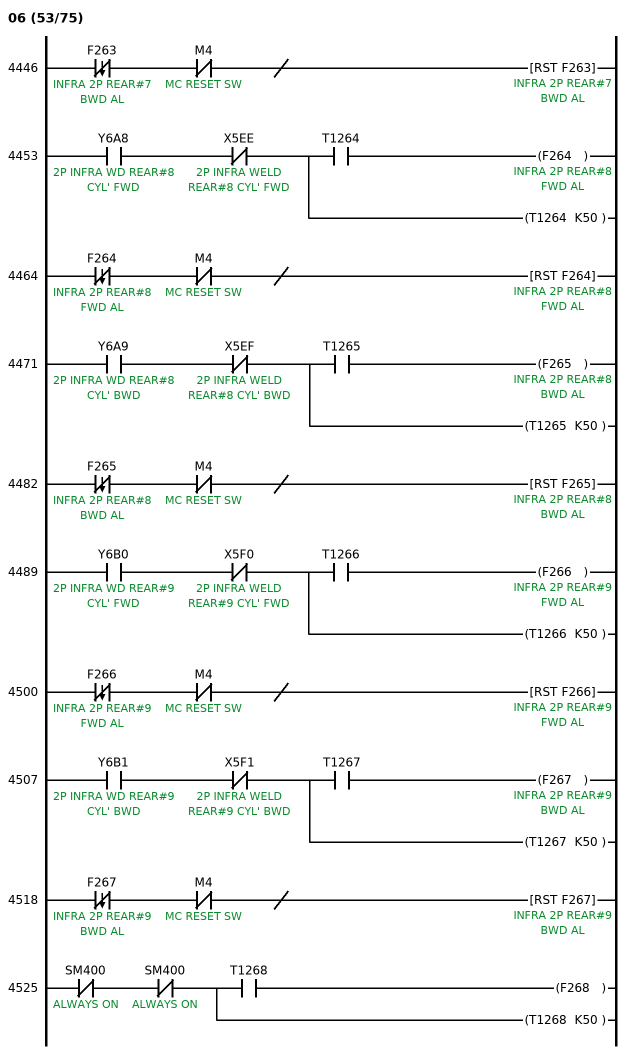
4446  LDFI    F263  ; INFRA 2P REAR#7 BWD AL
      ANI     M4  ; MC RESET SW
      INV
      RST     F263  ; INFRA 2P REAR#7 BWD AL
4453  LD      Y6A8  ; 2P INFRA WD REAR#8 CYL' FWD
      ANI     X5EE  ; 2P INFRA WELD REAR#8 CYL' FWD
      MPS
      AND     T1264
      OUT     F264  ; INFRA 2P REAR#8 FWD AL
      MPP
      OUT     T1264 K50
4464  LDFI    F264  ; INFRA 2P REAR#8 FWD AL
      ANI     M4  ; MC RESET SW
      INV
      RST     F264  ; INFRA 2P REAR#8 FWD AL
4471  LD      Y6A9  ; 2P INFRA WD REAR#8 CYL' BWD
      ANI     X5EF  ; 2P INFRA WELD REAR#8 CYL' BWD
      MPS
      AND     T1265
      OUT     F265  ; INFRA 2P REAR#8 BWD AL
      MPP
      OUT     T1265 K50
4482  LDFI    F265  ; INFRA 2P REAR#8 BWD AL
      ANI     M4  ; MC RESET SW
      INV
      RST     F265  ; INFRA 2P REAR#8 BWD AL
4489  LD      Y6B0  ; 2P INFRA WD REAR#9 CYL' FWD
      ANI     X5F0  ; 2P INFRA WELD REAR#9 CYL' FWD
      MPS
      AND     T1266
      OUT     F266  ; INFRA 2P REAR#9 FWD AL
      MPP
      OUT     T1266 K50
4500  LDFI    F266  ; INFRA 2P REAR#9 FWD AL
      ANI     M4  ; MC RESET SW
      INV
      RST     F266  ; INFRA 2P REAR#9 FWD AL
4507  LD      Y6B1  ; 2P INFRA WD REAR#9 CYL' BWD
      ANI     X5F1  ; 2P INFRA WELD REAR#9 CYL' BWD
      MPS
      AND     T1267
      OUT     F267  ; INFRA 2P REAR#9 BWD AL
      MPP
      OUT     T1267 K50
4518  LDFI    F267  ; INFRA 2P REAR#9 BWD AL
      ANI     M4  ; MC RESET SW
      INV
      RST     F267  ; INFRA 2P REAR#9 BWD AL
4525  LDI     SM400  ; ALWAYS ON
      ANI     SM400  ; ALWAYS ON
      MPS
      AND     T1268
      OUT     F268
      MPP
      OUT     T1268 K50
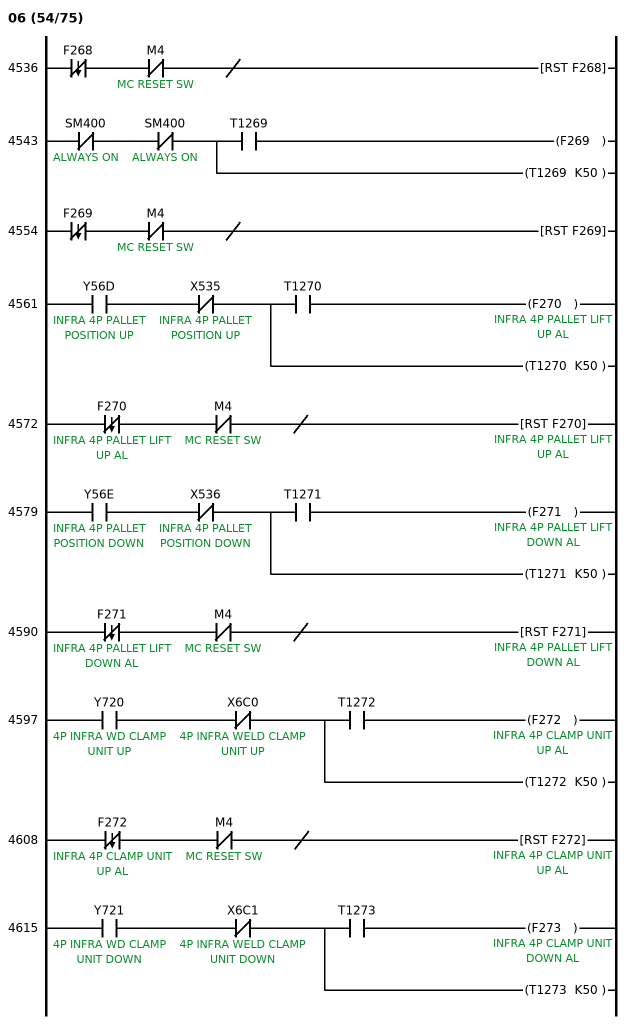
4536  LDFI    F268
      ANI     M4  ; MC RESET SW
      INV
      RST     F268
4543  LDI     SM400  ; ALWAYS ON
      ANI     SM400  ; ALWAYS ON
      MPS
      AND     T1269
      OUT     F269
      MPP
      OUT     T1269 K50
4554  LDFI    F269
      ANI     M4  ; MC RESET SW
      INV
      RST     F269
4561  LD      Y56D  ; INFRA 4P PALLET POSITION UP
      ANI     X535  ; INFRA 4P PALLET POSITION UP
      MPS
      AND     T1270
      OUT     F270  ; INFRA 4P PALLET LIFT UP AL
      MPP
      OUT     T1270 K50
4572  LDFI    F270  ; INFRA 4P PALLET LIFT UP AL
      ANI     M4  ; MC RESET SW
      INV
      RST     F270  ; INFRA 4P PALLET LIFT UP AL
4579  LD      Y56E  ; INFRA 4P PALLET POSITION DOWN
      ANI     X536  ; INFRA 4P PALLET POSITION DOWN
      MPS
      AND     T1271
      OUT     F271  ; INFRA 4P PALLET LIFT DOWN AL
      MPP
      OUT     T1271 K50
4590  LDFI    F271  ; INFRA 4P PALLET LIFT DOWN AL
      ANI     M4  ; MC RESET SW
      INV
      RST     F271  ; INFRA 4P PALLET LIFT DOWN AL
4597  LD      Y720  ; 4P INFRA WD CLAMP UNIT UP
      ANI     X6C0  ; 4P INFRA WELD CLAMP UNIT UP
      MPS
      AND     T1272
      OUT     F272  ; INFRA 4P CLAMP UNIT UP AL
      MPP
      OUT     T1272 K50
4608  LDFI    F272  ; INFRA 4P CLAMP UNIT UP AL
      ANI     M4  ; MC RESET SW
      INV
      RST     F272  ; INFRA 4P CLAMP UNIT UP AL
4615  LD      Y721  ; 4P INFRA WD CLAMP UNIT DOWN
      ANI     X6C1  ; 4P INFRA WELD CLAMP UNIT DOWN
      MPS
      AND     T1273
      OUT     F273  ; INFRA 4P CLAMP UNIT DOWN AL
      MPP
      OUT     T1273 K50
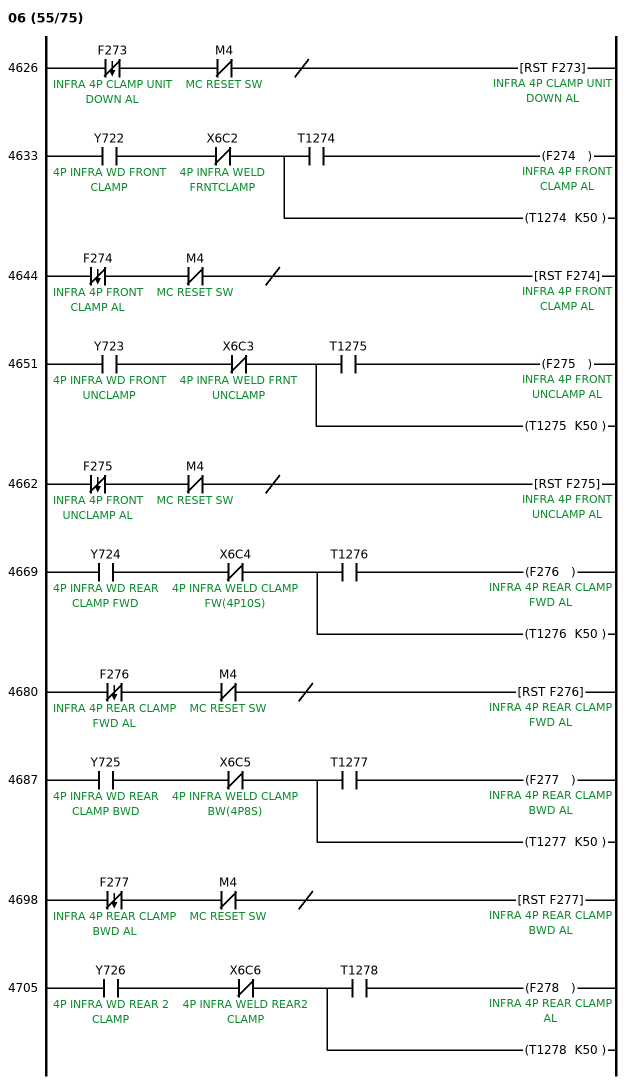
4626  LDFI    F273  ; INFRA 4P CLAMP UNIT DOWN AL
      ANI     M4  ; MC RESET SW
      INV
      RST     F273  ; INFRA 4P CLAMP UNIT DOWN AL
4633  LD      Y722  ; 4P INFRA WD FRONT CLAMP
      ANI     X6C2  ; 4P INFRA WELD FRNTCLAMP
      MPS
      AND     T1274
      OUT     F274  ; INFRA 4P FRONT CLAMP AL
      MPP
      OUT     T1274 K50
4644  LDFI    F274  ; INFRA 4P FRONT CLAMP AL
      ANI     M4  ; MC RESET SW
      INV
      RST     F274  ; INFRA 4P FRONT CLAMP AL
4651  LD      Y723  ; 4P INFRA WD FRONT UNCLAMP
      ANI     X6C3  ; 4P INFRA WELD FRNT UNCLAMP
      MPS
      AND     T1275
      OUT     F275  ; INFRA 4P FRONT UNCLAMP AL
      MPP
      OUT     T1275 K50
4662  LDFI    F275  ; INFRA 4P FRONT UNCLAMP AL
      ANI     M4  ; MC RESET SW
      INV
      RST     F275  ; INFRA 4P FRONT UNCLAMP AL
4669  LD      Y724  ; 4P INFRA WD REAR CLAMP FWD
      ANI     X6C4  ; 4P INFRA WELD CLAMP FW(4P10S)
      MPS
      AND     T1276
      OUT     F276  ; INFRA 4P REAR CLAMP FWD AL
      MPP
      OUT     T1276 K50
4680  LDFI    F276  ; INFRA 4P REAR CLAMP FWD AL
      ANI     M4  ; MC RESET SW
      INV
      RST     F276  ; INFRA 4P REAR CLAMP FWD AL
4687  LD      Y725  ; 4P INFRA WD REAR CLAMP BWD
      ANI     X6C5  ; 4P INFRA WELD CLAMP BW(4P8S)
      MPS
      AND     T1277
      OUT     F277  ; INFRA 4P REAR CLAMP BWD AL
      MPP
      OUT     T1277 K50
4698  LDFI    F277  ; INFRA 4P REAR CLAMP BWD AL
      ANI     M4  ; MC RESET SW
      INV
      RST     F277  ; INFRA 4P REAR CLAMP BWD AL
4705  LD      Y726  ; 4P INFRA WD REAR 2 CLAMP
      ANI     X6C6  ; 4P INFRA WELD REAR2 CLAMP
      MPS
      AND     T1278
      OUT     F278  ; INFRA 4P REAR CLAMP AL
      MPP
      OUT     T1278 K50
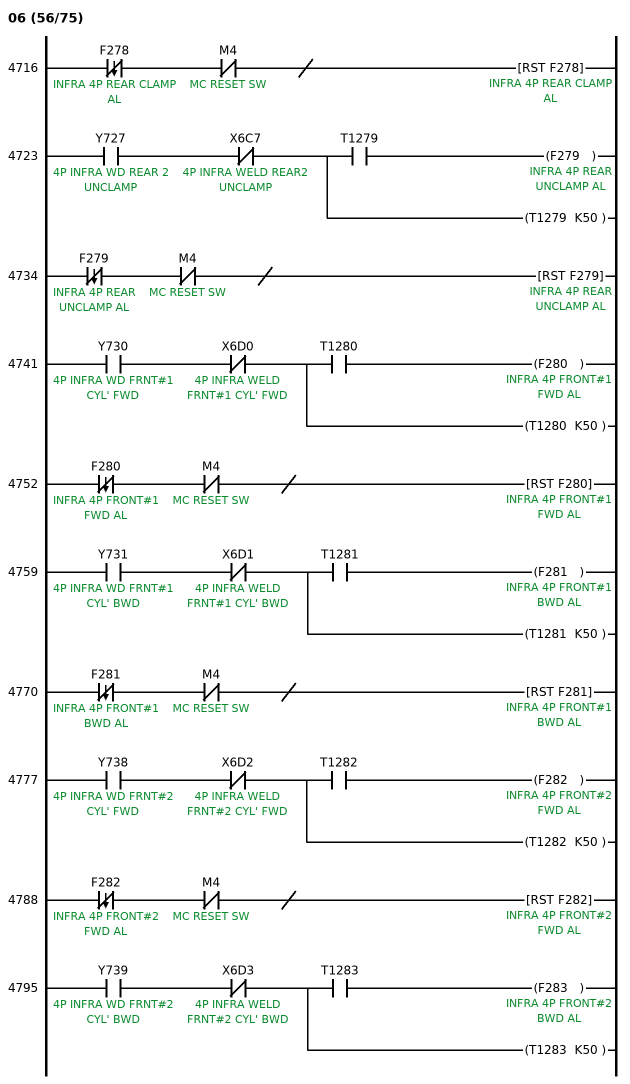
4716  LDFI    F278  ; INFRA 4P REAR CLAMP AL
      ANI     M4  ; MC RESET SW
      INV
      RST     F278  ; INFRA 4P REAR CLAMP AL
4723  LD      Y727  ; 4P INFRA WD REAR 2 UNCLAMP
      ANI     X6C7  ; 4P INFRA WELD REAR2 UNCLAMP
      MPS
      AND     T1279
      OUT     F279  ; INFRA 4P REAR UNCLAMP AL
      MPP
      OUT     T1279 K50
4734  LDFI    F279  ; INFRA 4P REAR UNCLAMP AL
      ANI     M4  ; MC RESET SW
      INV
      RST     F279  ; INFRA 4P REAR UNCLAMP AL
4741  LD      Y730  ; 4P INFRA WD FRNT#1 CYL' FWD
      ANI     X6D0  ; 4P INFRA WELD FRNT#1 CYL' FWD
      MPS
      AND     T1280
      OUT     F280  ; INFRA 4P FRONT#1 FWD AL
      MPP
      OUT     T1280 K50
4752  LDFI    F280  ; INFRA 4P FRONT#1 FWD AL
      ANI     M4  ; MC RESET SW
      INV
      RST     F280  ; INFRA 4P FRONT#1 FWD AL
4759  LD      Y731  ; 4P INFRA WD FRNT#1 CYL' BWD
      ANI     X6D1  ; 4P INFRA WELD FRNT#1 CYL' BWD
      MPS
      AND     T1281
      OUT     F281  ; INFRA 4P FRONT#1 BWD AL
      MPP
      OUT     T1281 K50
4770  LDFI    F281  ; INFRA 4P FRONT#1 BWD AL
      ANI     M4  ; MC RESET SW
      INV
      RST     F281  ; INFRA 4P FRONT#1 BWD AL
4777  LD      Y738  ; 4P INFRA WD FRNT#2 CYL' FWD
      ANI     X6D2  ; 4P INFRA WELD FRNT#2 CYL' FWD
      MPS
      AND     T1282
      OUT     F282  ; INFRA 4P FRONT#2 FWD AL
      MPP
      OUT     T1282 K50
4788  LDFI    F282  ; INFRA 4P FRONT#2 FWD AL
      ANI     M4  ; MC RESET SW
      INV
      RST     F282  ; INFRA 4P FRONT#2 FWD AL
4795  LD      Y739  ; 4P INFRA WD FRNT#2 CYL' BWD
      ANI     X6D3  ; 4P INFRA WELD FRNT#2 CYL' BWD
      MPS
      AND     T1283
      OUT     F283  ; INFRA 4P FRONT#2 BWD AL
      MPP
      OUT     T1283 K50
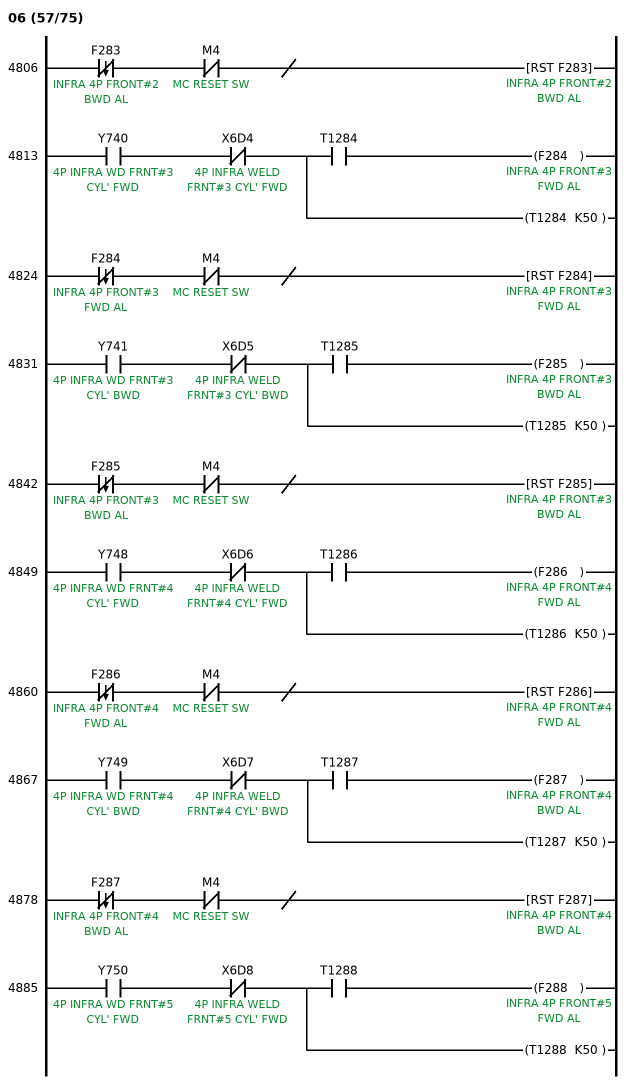
4806  LDFI    F283  ; INFRA 4P FRONT#2 BWD AL
      ANI     M4  ; MC RESET SW
      INV
      RST     F283  ; INFRA 4P FRONT#2 BWD AL
4813  LD      Y740  ; 4P INFRA WD FRNT#3 CYL' FWD
      ANI     X6D4  ; 4P INFRA WELD FRNT#3 CYL' FWD
      MPS
      AND     T1284
      OUT     F284  ; INFRA 4P FRONT#3 FWD AL
      MPP
      OUT     T1284 K50
4824  LDFI    F284  ; INFRA 4P FRONT#3 FWD AL
      ANI     M4  ; MC RESET SW
      INV
      RST     F284  ; INFRA 4P FRONT#3 FWD AL
4831  LD      Y741  ; 4P INFRA WD FRNT#3 CYL' BWD
      ANI     X6D5  ; 4P INFRA WELD FRNT#3 CYL' BWD
      MPS
      AND     T1285
      OUT     F285  ; INFRA 4P FRONT#3 BWD AL
      MPP
      OUT     T1285 K50
4842  LDFI    F285  ; INFRA 4P FRONT#3 BWD AL
      ANI     M4  ; MC RESET SW
      INV
      RST     F285  ; INFRA 4P FRONT#3 BWD AL
4849  LD      Y748  ; 4P INFRA WD FRNT#4 CYL' FWD
      ANI     X6D6  ; 4P INFRA WELD FRNT#4 CYL' FWD
      MPS
      AND     T1286
      OUT     F286  ; INFRA 4P FRONT#4 FWD AL
      MPP
      OUT     T1286 K50
4860  LDFI    F286  ; INFRA 4P FRONT#4 FWD AL
      ANI     M4  ; MC RESET SW
      INV
      RST     F286  ; INFRA 4P FRONT#4 FWD AL
4867  LD      Y749  ; 4P INFRA WD FRNT#4 CYL' BWD
      ANI     X6D7  ; 4P INFRA WELD FRNT#4 CYL' BWD
      MPS
      AND     T1287
      OUT     F287  ; INFRA 4P FRONT#4 BWD AL
      MPP
      OUT     T1287 K50
4878  LDFI    F287  ; INFRA 4P FRONT#4 BWD AL
      ANI     M4  ; MC RESET SW
      INV
      RST     F287  ; INFRA 4P FRONT#4 BWD AL
4885  LD      Y750  ; 4P INFRA WD FRNT#5 CYL' FWD
      ANI     X6D8  ; 4P INFRA WELD FRNT#5 CYL' FWD
      MPS
      AND     T1288
      OUT     F288  ; INFRA 4P FRONT#5 FWD AL
      MPP
      OUT     T1288 K50
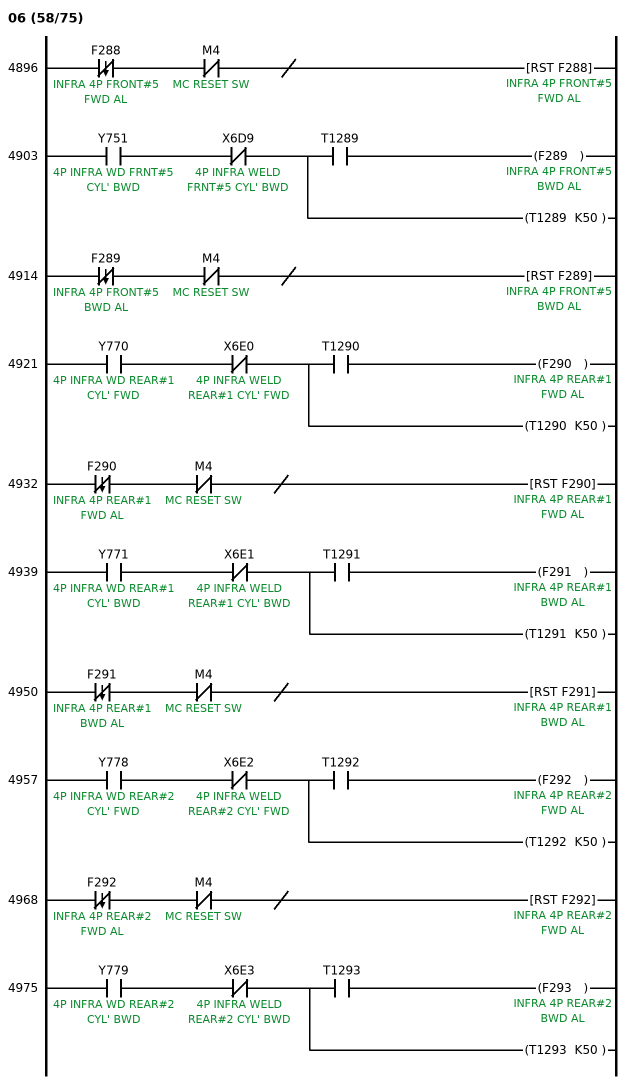
4896  LDFI    F288  ; INFRA 4P FRONT#5 FWD AL
      ANI     M4  ; MC RESET SW
      INV
      RST     F288  ; INFRA 4P FRONT#5 FWD AL
4903  LD      Y751  ; 4P INFRA WD FRNT#5 CYL' BWD
      ANI     X6D9  ; 4P INFRA WELD FRNT#5 CYL' BWD
      MPS
      AND     T1289
      OUT     F289  ; INFRA 4P FRONT#5 BWD AL
      MPP
      OUT     T1289 K50
4914  LDFI    F289  ; INFRA 4P FRONT#5 BWD AL
      ANI     M4  ; MC RESET SW
      INV
      RST     F289  ; INFRA 4P FRONT#5 BWD AL
4921  LD      Y770  ; 4P INFRA WD REAR#1 CYL' FWD
      ANI     X6E0  ; 4P INFRA WELD REAR#1 CYL' FWD
      MPS
      AND     T1290
      OUT     F290  ; INFRA 4P REAR#1 FWD AL
      MPP
      OUT     T1290 K50
4932  LDFI    F290  ; INFRA 4P REAR#1 FWD AL
      ANI     M4  ; MC RESET SW
      INV
      RST     F290  ; INFRA 4P REAR#1 FWD AL
4939  LD      Y771  ; 4P INFRA WD REAR#1 CYL' BWD
      ANI     X6E1  ; 4P INFRA WELD REAR#1 CYL' BWD
      MPS
      AND     T1291
      OUT     F291  ; INFRA 4P REAR#1 BWD AL
      MPP
      OUT     T1291 K50
4950  LDFI    F291  ; INFRA 4P REAR#1 BWD AL
      ANI     M4  ; MC RESET SW
      INV
      RST     F291  ; INFRA 4P REAR#1 BWD AL
4957  LD      Y778  ; 4P INFRA WD REAR#2 CYL' FWD
      ANI     X6E2  ; 4P INFRA WELD REAR#2 CYL' FWD
      MPS
      AND     T1292
      OUT     F292  ; INFRA 4P REAR#2 FWD AL
      MPP
      OUT     T1292 K50
4968  LDFI    F292  ; INFRA 4P REAR#2 FWD AL
      ANI     M4  ; MC RESET SW
      INV
      RST     F292  ; INFRA 4P REAR#2 FWD AL
4975  LD      Y779  ; 4P INFRA WD REAR#2 CYL' BWD
      ANI     X6E3  ; 4P INFRA WELD REAR#2 CYL' BWD
      MPS
      AND     T1293
      OUT     F293  ; INFRA 4P REAR#2 BWD AL
      MPP
      OUT     T1293 K50
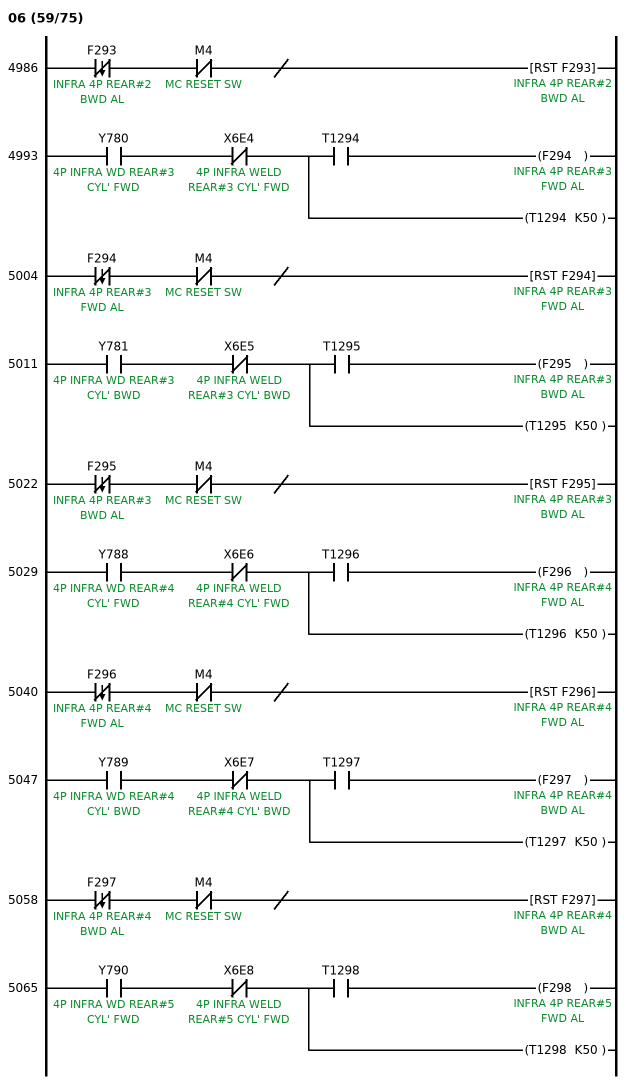
4986  LDFI    F293  ; INFRA 4P REAR#2 BWD AL
      ANI     M4  ; MC RESET SW
      INV
      RST     F293  ; INFRA 4P REAR#2 BWD AL
4993  LD      Y780  ; 4P INFRA WD REAR#3 CYL' FWD
      ANI     X6E4  ; 4P INFRA WELD REAR#3 CYL' FWD
      MPS
      AND     T1294
      OUT     F294  ; INFRA 4P REAR#3 FWD AL
      MPP
      OUT     T1294 K50
5004  LDFI    F294  ; INFRA 4P REAR#3 FWD AL
      ANI     M4  ; MC RESET SW
      INV
      RST     F294  ; INFRA 4P REAR#3 FWD AL
5011  LD      Y781  ; 4P INFRA WD REAR#3 CYL' BWD
      ANI     X6E5  ; 4P INFRA WELD REAR#3 CYL' BWD
      MPS
      AND     T1295
      OUT     F295  ; INFRA 4P REAR#3 BWD AL
      MPP
      OUT     T1295 K50
5022  LDFI    F295  ; INFRA 4P REAR#3 BWD AL
      ANI     M4  ; MC RESET SW
      INV
      RST     F295  ; INFRA 4P REAR#3 BWD AL
5029  LD      Y788  ; 4P INFRA WD REAR#4 CYL' FWD
      ANI     X6E6  ; 4P INFRA WELD REAR#4 CYL' FWD
      MPS
      AND     T1296
      OUT     F296  ; INFRA 4P REAR#4 FWD AL
      MPP
      OUT     T1296 K50
5040  LDFI    F296  ; INFRA 4P REAR#4 FWD AL
      ANI     M4  ; MC RESET SW
      INV
      RST     F296  ; INFRA 4P REAR#4 FWD AL
5047  LD      Y789  ; 4P INFRA WD REAR#4 CYL' BWD
      ANI     X6E7  ; 4P INFRA WELD REAR#4 CYL' BWD
      MPS
      AND     T1297
      OUT     F297  ; INFRA 4P REAR#4 BWD AL
      MPP
      OUT     T1297 K50
5058  LDFI    F297  ; INFRA 4P REAR#4 BWD AL
      ANI     M4  ; MC RESET SW
      INV
      RST     F297  ; INFRA 4P REAR#4 BWD AL
5065  LD      Y790  ; 4P INFRA WD REAR#5 CYL' FWD
      ANI     X6E8  ; 4P INFRA WELD REAR#5 CYL' FWD
      MPS
      AND     T1298
      OUT     F298  ; INFRA 4P REAR#5 FWD AL
      MPP
      OUT     T1298 K50
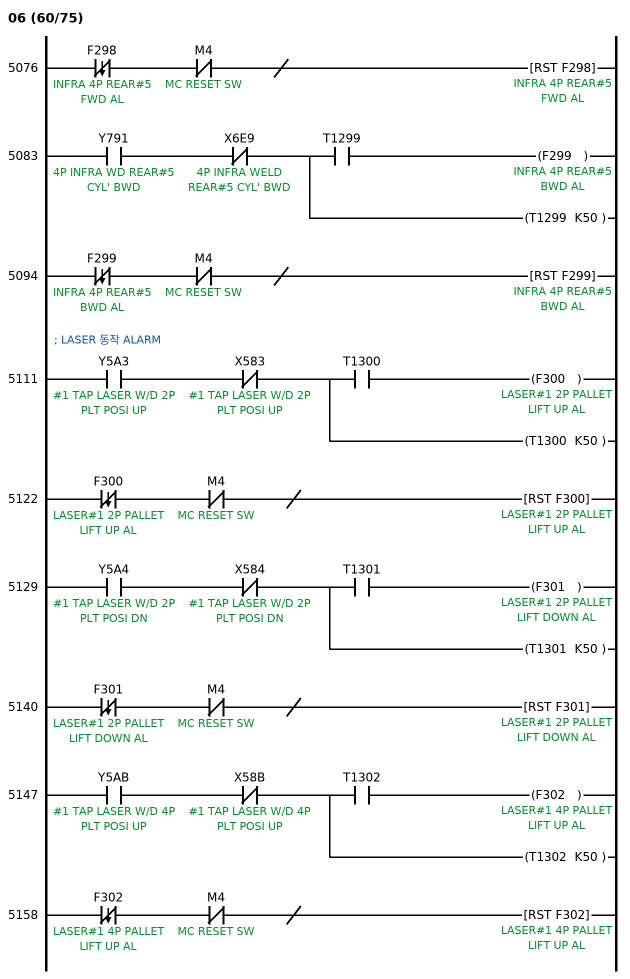
5076  LDFI    F298  ; INFRA 4P REAR#5 FWD AL
      ANI     M4  ; MC RESET SW
      INV
      RST     F298  ; INFRA 4P REAR#5 FWD AL
5083  LD      Y791  ; 4P INFRA WD REAR#5 CYL' BWD
      ANI     X6E9  ; 4P INFRA WELD REAR#5 CYL' BWD
      MPS
      AND     T1299
      OUT     F299  ; INFRA 4P REAR#5 BWD AL
      MPP
      OUT     T1299 K50
5094  LDFI    F299  ; INFRA 4P REAR#5 BWD AL
      ANI     M4  ; MC RESET SW
      INV
      RST     F299  ; INFRA 4P REAR#5 BWD AL
; LASER 동작 ALARM
5111  LD      Y5A3  ; #1 TAP LASER W/D 2P PLT POSI UP
      ANI     X583  ; #1 TAP LASER W/D 2P PLT POSI UP
      MPS
      AND     T1300
      OUT     F300  ; LASER#1 2P PALLET LIFT UP AL
      MPP
      OUT     T1300 K50
5122  LDFI    F300  ; LASER#1 2P PALLET LIFT UP AL
      ANI     M4  ; MC RESET SW
      INV
      RST     F300  ; LASER#1 2P PALLET LIFT UP AL
5129  LD      Y5A4  ; #1 TAP LASER W/D 2P PLT POSI DN
      ANI     X584  ; #1 TAP LASER W/D 2P PLT POSI DN
      MPS
      AND     T1301
      OUT     F301  ; LASER#1 2P PALLET LIFT DOWN AL
      MPP
      OUT     T1301 K50
5140  LDFI    F301  ; LASER#1 2P PALLET LIFT DOWN AL
      ANI     M4  ; MC RESET SW
      INV
      RST     F301  ; LASER#1 2P PALLET LIFT DOWN AL
5147  LD      Y5AB  ; #1 TAP LASER W/D 4P PLT POSI UP
      ANI     X58B  ; #1 TAP LASER W/D 4P PLT POSI UP
      MPS
      AND     T1302
      OUT     F302  ; LASER#1 4P PALLET LIFT UP AL
      MPP
      OUT     T1302 K50
5158  LDFI    F302  ; LASER#1 4P PALLET LIFT UP AL
      ANI     M4  ; MC RESET SW
      INV
      RST     F302  ; LASER#1 4P PALLET LIFT UP AL
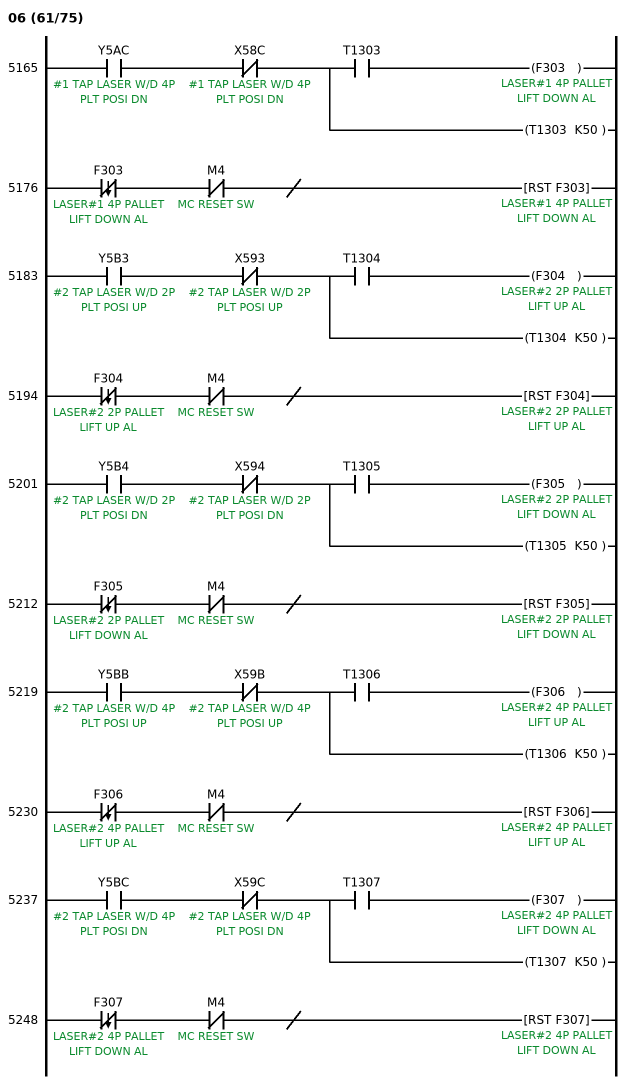
5165  LD      Y5AC  ; #1 TAP LASER W/D 4P PLT POSI DN
      ANI     X58C  ; #1 TAP LASER W/D 4P PLT POSI DN
      MPS
      AND     T1303
      OUT     F303  ; LASER#1 4P PALLET LIFT DOWN AL
      MPP
      OUT     T1303 K50
5176  LDFI    F303  ; LASER#1 4P PALLET LIFT DOWN AL
      ANI     M4  ; MC RESET SW
      INV
      RST     F303  ; LASER#1 4P PALLET LIFT DOWN AL
5183  LD      Y5B3  ; #2 TAP LASER W/D 2P PLT POSI UP
      ANI     X593  ; #2 TAP LASER W/D 2P PLT POSI UP
      MPS
      AND     T1304
      OUT     F304  ; LASER#2 2P PALLET LIFT UP AL
      MPP
      OUT     T1304 K50
5194  LDFI    F304  ; LASER#2 2P PALLET LIFT UP AL
      ANI     M4  ; MC RESET SW
      INV
      RST     F304  ; LASER#2 2P PALLET LIFT UP AL
5201  LD      Y5B4  ; #2 TAP LASER W/D 2P PLT POSI DN
      ANI     X594  ; #2 TAP LASER W/D 2P PLT POSI DN
      MPS
      AND     T1305
      OUT     F305  ; LASER#2 2P PALLET LIFT DOWN AL
      MPP
      OUT     T1305 K50
5212  LDFI    F305  ; LASER#2 2P PALLET LIFT DOWN AL
      ANI     M4  ; MC RESET SW
      INV
      RST     F305  ; LASER#2 2P PALLET LIFT DOWN AL
5219  LD      Y5BB  ; #2 TAP LASER W/D 4P PLT POSI UP
      ANI     X59B  ; #2 TAP LASER W/D 4P PLT POSI UP
      MPS
      AND     T1306
      OUT     F306  ; LASER#2 4P PALLET LIFT UP AL
      MPP
      OUT     T1306 K50
5230  LDFI    F306  ; LASER#2 4P PALLET LIFT UP AL
      ANI     M4  ; MC RESET SW
      INV
      RST     F306  ; LASER#2 4P PALLET LIFT UP AL
5237  LD      Y5BC  ; #2 TAP LASER W/D 4P PLT POSI DN
      ANI     X59C  ; #2 TAP LASER W/D 4P PLT POSI DN
      MPS
      AND     T1307
      OUT     F307  ; LASER#2 4P PALLET LIFT DOWN AL
      MPP
      OUT     T1307 K50
5248  LDFI    F307  ; LASER#2 4P PALLET LIFT DOWN AL
      ANI     M4  ; MC RESET SW
      INV
      RST     F307  ; LASER#2 4P PALLET LIFT DOWN AL
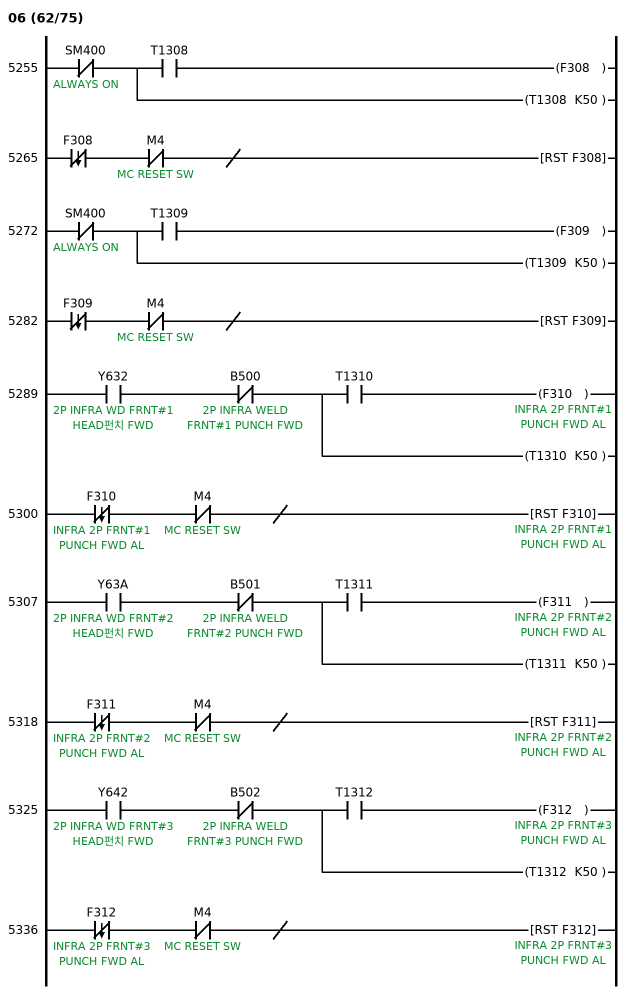
5255  LDI     SM400  ; ALWAYS ON
      MPS
      AND     T1308
      OUT     F308
      MPP
      OUT     T1308 K50
5265  LDFI    F308
      ANI     M4  ; MC RESET SW
      INV
      RST     F308
5272  LDI     SM400  ; ALWAYS ON
      MPS
      AND     T1309
      OUT     F309
      MPP
      OUT     T1309 K50
5282  LDFI    F309
      ANI     M4  ; MC RESET SW
      INV
      RST     F309
5289  LD      Y632  ; 2P INFRA WD FRNT#1 HEAD펀치 FWD
      ANI     B500  ; 2P INFRA WELD FRNT#1 PUNCH FWD
      MPS
      AND     T1310
      OUT     F310  ; INFRA 2P FRNT#1 PUNCH FWD AL
      MPP
      OUT     T1310 K50
5300  LDFI    F310  ; INFRA 2P FRNT#1 PUNCH FWD AL
      ANI     M4  ; MC RESET SW
      INV
      RST     F310  ; INFRA 2P FRNT#1 PUNCH FWD AL
5307  LD      Y63A  ; 2P INFRA WD FRNT#2 HEAD펀치 FWD
      ANI     B501  ; 2P INFRA WELD FRNT#2 PUNCH FWD
      MPS
      AND     T1311
      OUT     F311  ; INFRA 2P FRNT#2 PUNCH FWD AL
      MPP
      OUT     T1311 K50
5318  LDFI    F311  ; INFRA 2P FRNT#2 PUNCH FWD AL
      ANI     M4  ; MC RESET SW
      INV
      RST     F311  ; INFRA 2P FRNT#2 PUNCH FWD AL
5325  LD      Y642  ; 2P INFRA WD FRNT#3 HEAD펀치 FWD
      ANI     B502  ; 2P INFRA WELD FRNT#3 PUNCH FWD
      MPS
      AND     T1312
      OUT     F312  ; INFRA 2P FRNT#3 PUNCH FWD AL
      MPP
      OUT     T1312 K50
5336  LDFI    F312  ; INFRA 2P FRNT#3 PUNCH FWD AL
      ANI     M4  ; MC RESET SW
      INV
      RST     F312  ; INFRA 2P FRNT#3 PUNCH FWD AL
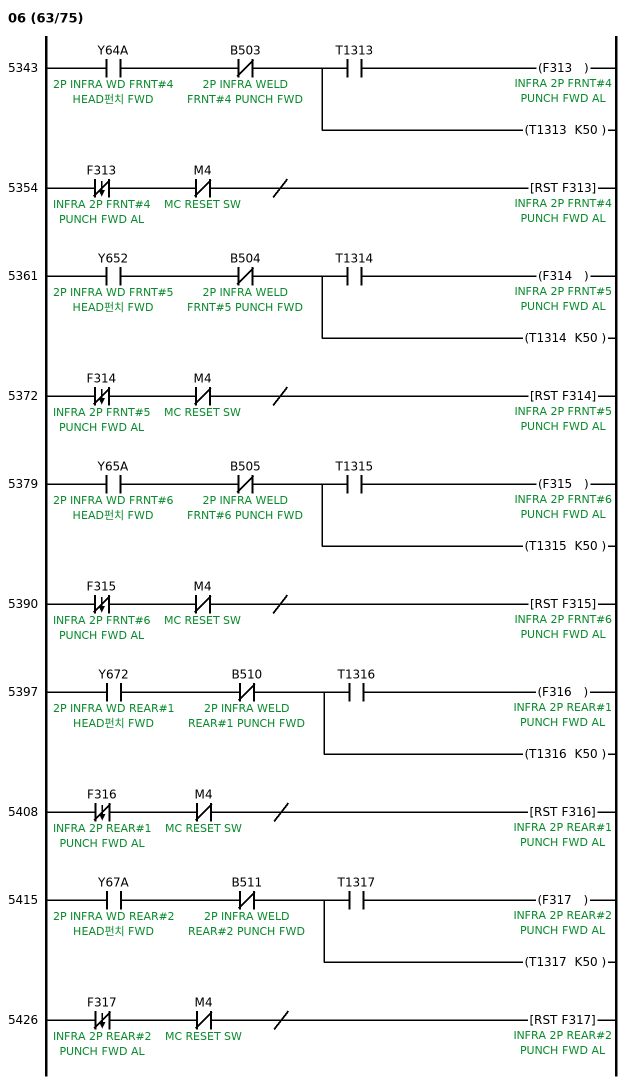
5343  LD      Y64A  ; 2P INFRA WD FRNT#4 HEAD펀치 FWD
      ANI     B503  ; 2P INFRA WELD FRNT#4 PUNCH FWD
      MPS
      AND     T1313
      OUT     F313  ; INFRA 2P FRNT#4 PUNCH FWD AL
      MPP
      OUT     T1313 K50
5354  LDFI    F313  ; INFRA 2P FRNT#4 PUNCH FWD AL
      ANI     M4  ; MC RESET SW
      INV
      RST     F313  ; INFRA 2P FRNT#4 PUNCH FWD AL
5361  LD      Y652  ; 2P INFRA WD FRNT#5 HEAD펀치 FWD
      ANI     B504  ; 2P INFRA WELD FRNT#5 PUNCH FWD
      MPS
      AND     T1314
      OUT     F314  ; INFRA 2P FRNT#5 PUNCH FWD AL
      MPP
      OUT     T1314 K50
5372  LDFI    F314  ; INFRA 2P FRNT#5 PUNCH FWD AL
      ANI     M4  ; MC RESET SW
      INV
      RST     F314  ; INFRA 2P FRNT#5 PUNCH FWD AL
5379  LD      Y65A  ; 2P INFRA WD FRNT#6 HEAD펀치 FWD
      ANI     B505  ; 2P INFRA WELD FRNT#6 PUNCH FWD
      MPS
      AND     T1315
      OUT     F315  ; INFRA 2P FRNT#6 PUNCH FWD AL
      MPP
      OUT     T1315 K50
5390  LDFI    F315  ; INFRA 2P FRNT#6 PUNCH FWD AL
      ANI     M4  ; MC RESET SW
      INV
      RST     F315  ; INFRA 2P FRNT#6 PUNCH FWD AL
5397  LD      Y672  ; 2P INFRA WD REAR#1 HEAD펀치 FWD
      ANI     B510  ; 2P INFRA WELD REAR#1 PUNCH FWD
      MPS
      AND     T1316
      OUT     F316  ; INFRA 2P REAR#1 PUNCH FWD AL
      MPP
      OUT     T1316 K50
5408  LDFI    F316  ; INFRA 2P REAR#1 PUNCH FWD AL
      ANI     M4  ; MC RESET SW
      INV
      RST     F316  ; INFRA 2P REAR#1 PUNCH FWD AL
5415  LD      Y67A  ; 2P INFRA WD REAR#2 HEAD펀치 FWD
      ANI     B511  ; 2P INFRA WELD REAR#2 PUNCH FWD
      MPS
      AND     T1317
      OUT     F317  ; INFRA 2P REAR#2 PUNCH FWD AL
      MPP
      OUT     T1317 K50
5426  LDFI    F317  ; INFRA 2P REAR#2 PUNCH FWD AL
      ANI     M4  ; MC RESET SW
      INV
      RST     F317  ; INFRA 2P REAR#2 PUNCH FWD AL
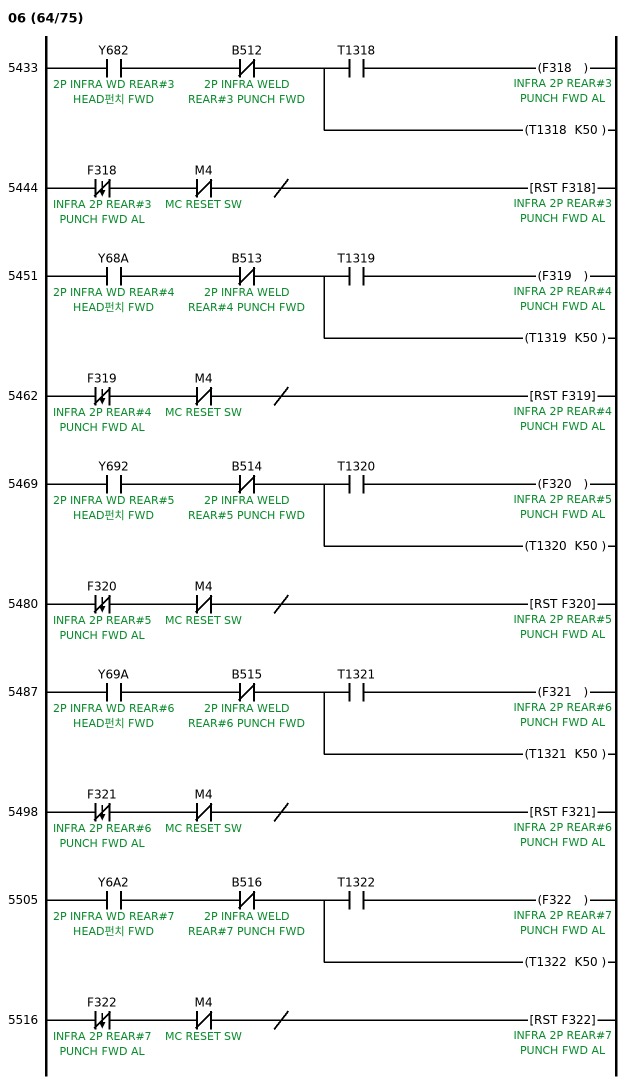
5433  LD      Y682  ; 2P INFRA WD REAR#3 HEAD펀치 FWD
      ANI     B512  ; 2P INFRA WELD REAR#3 PUNCH FWD
      MPS
      AND     T1318
      OUT     F318  ; INFRA 2P REAR#3 PUNCH FWD AL
      MPP
      OUT     T1318 K50
5444  LDFI    F318  ; INFRA 2P REAR#3 PUNCH FWD AL
      ANI     M4  ; MC RESET SW
      INV
      RST     F318  ; INFRA 2P REAR#3 PUNCH FWD AL
5451  LD      Y68A  ; 2P INFRA WD REAR#4 HEAD펀치 FWD
      ANI     B513  ; 2P INFRA WELD REAR#4 PUNCH FWD
      MPS
      AND     T1319
      OUT     F319  ; INFRA 2P REAR#4 PUNCH FWD AL
      MPP
      OUT     T1319 K50
5462  LDFI    F319  ; INFRA 2P REAR#4 PUNCH FWD AL
      ANI     M4  ; MC RESET SW
      INV
      RST     F319  ; INFRA 2P REAR#4 PUNCH FWD AL
5469  LD      Y692  ; 2P INFRA WD REAR#5 HEAD펀치 FWD
      ANI     B514  ; 2P INFRA WELD REAR#5 PUNCH FWD
      MPS
      AND     T1320
      OUT     F320  ; INFRA 2P REAR#5 PUNCH FWD AL
      MPP
      OUT     T1320 K50
5480  LDFI    F320  ; INFRA 2P REAR#5 PUNCH FWD AL
      ANI     M4  ; MC RESET SW
      INV
      RST     F320  ; INFRA 2P REAR#5 PUNCH FWD AL
5487  LD      Y69A  ; 2P INFRA WD REAR#6 HEAD펀치 FWD
      ANI     B515  ; 2P INFRA WELD REAR#6 PUNCH FWD
      MPS
      AND     T1321
      OUT     F321  ; INFRA 2P REAR#6 PUNCH FWD AL
      MPP
      OUT     T1321 K50
5498  LDFI    F321  ; INFRA 2P REAR#6 PUNCH FWD AL
      ANI     M4  ; MC RESET SW
      INV
      RST     F321  ; INFRA 2P REAR#6 PUNCH FWD AL
5505  LD      Y6A2  ; 2P INFRA WD REAR#7 HEAD펀치 FWD
      ANI     B516  ; 2P INFRA WELD REAR#7 PUNCH FWD
      MPS
      AND     T1322
      OUT     F322  ; INFRA 2P REAR#7 PUNCH FWD AL
      MPP
      OUT     T1322 K50
5516  LDFI    F322  ; INFRA 2P REAR#7 PUNCH FWD AL
      ANI     M4  ; MC RESET SW
      INV
      RST     F322  ; INFRA 2P REAR#7 PUNCH FWD AL
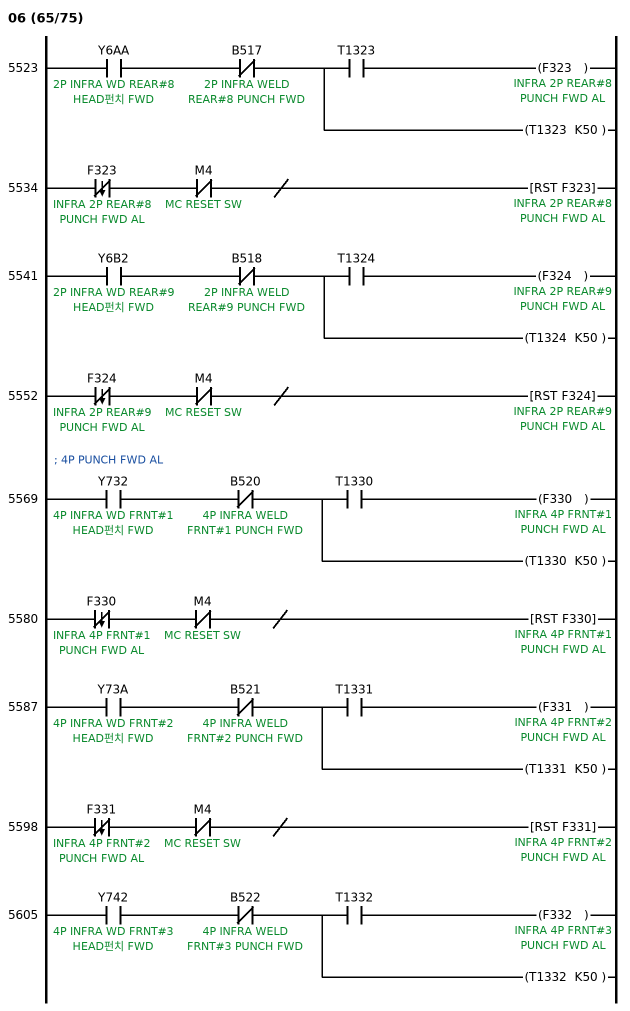
5523  LD      Y6AA  ; 2P INFRA WD REAR#8 HEAD펀치 FWD
      ANI     B517  ; 2P INFRA WELD REAR#8 PUNCH FWD
      MPS
      AND     T1323
      OUT     F323  ; INFRA 2P REAR#8 PUNCH FWD AL
      MPP
      OUT     T1323 K50
5534  LDFI    F323  ; INFRA 2P REAR#8 PUNCH FWD AL
      ANI     M4  ; MC RESET SW
      INV
      RST     F323  ; INFRA 2P REAR#8 PUNCH FWD AL
5541  LD      Y6B2  ; 2P INFRA WD REAR#9 HEAD펀치 FWD
      ANI     B518  ; 2P INFRA WELD REAR#9 PUNCH FWD
      MPS
      AND     T1324
      OUT     F324  ; INFRA 2P REAR#9 PUNCH FWD AL
      MPP
      OUT     T1324 K50
5552  LDFI    F324  ; INFRA 2P REAR#9 PUNCH FWD AL
      ANI     M4  ; MC RESET SW
      INV
      RST     F324  ; INFRA 2P REAR#9 PUNCH FWD AL
; 4P PUNCH FWD AL
5569  LD      Y732  ; 4P INFRA WD FRNT#1 HEAD펀치 FWD
      ANI     B520  ; 4P INFRA WELD FRNT#1 PUNCH FWD
      MPS
      AND     T1330
      OUT     F330  ; INFRA 4P FRNT#1 PUNCH FWD AL
      MPP
      OUT     T1330 K50
5580  LDFI    F330  ; INFRA 4P FRNT#1 PUNCH FWD AL
      ANI     M4  ; MC RESET SW
      INV
      RST     F330  ; INFRA 4P FRNT#1 PUNCH FWD AL
5587  LD      Y73A  ; 4P INFRA WD FRNT#2 HEAD펀치 FWD
      ANI     B521  ; 4P INFRA WELD FRNT#2 PUNCH FWD
      MPS
      AND     T1331
      OUT     F331  ; INFRA 4P FRNT#2 PUNCH FWD AL
      MPP
      OUT     T1331 K50
5598  LDFI    F331  ; INFRA 4P FRNT#2 PUNCH FWD AL
      ANI     M4  ; MC RESET SW
      INV
      RST     F331  ; INFRA 4P FRNT#2 PUNCH FWD AL
5605  LD      Y742  ; 4P INFRA WD FRNT#3 HEAD펀치 FWD
      ANI     B522  ; 4P INFRA WELD FRNT#3 PUNCH FWD
      MPS
      AND     T1332
      OUT     F332  ; INFRA 4P FRNT#3 PUNCH FWD AL
      MPP
      OUT     T1332 K50
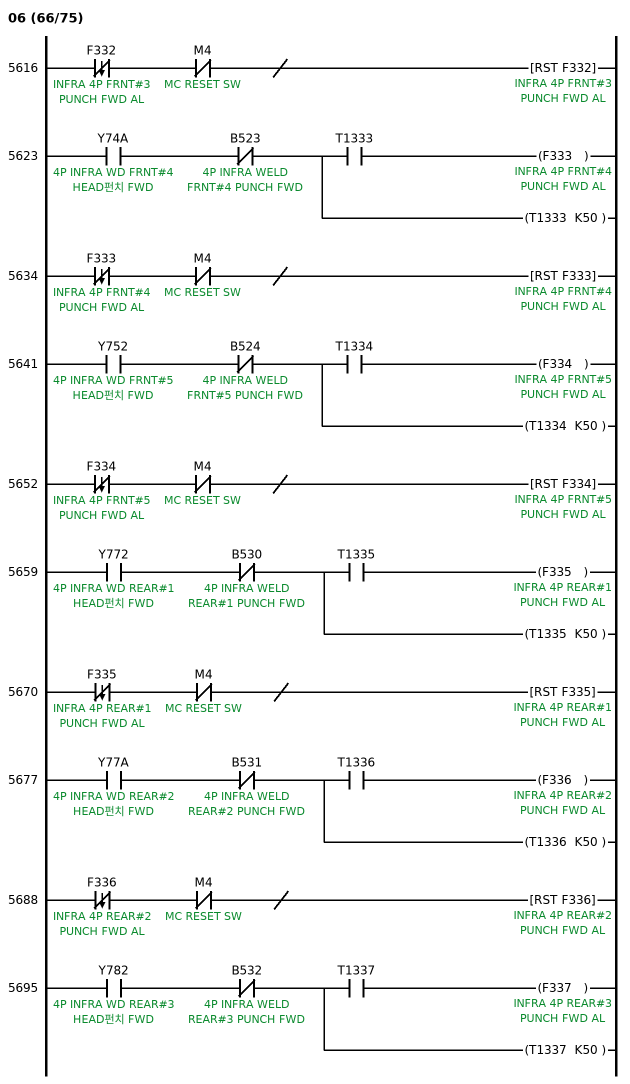
5616  LDFI    F332  ; INFRA 4P FRNT#3 PUNCH FWD AL
      ANI     M4  ; MC RESET SW
      INV
      RST     F332  ; INFRA 4P FRNT#3 PUNCH FWD AL
5623  LD      Y74A  ; 4P INFRA WD FRNT#4 HEAD펀치 FWD
      ANI     B523  ; 4P INFRA WELD FRNT#4 PUNCH FWD
      MPS
      AND     T1333
      OUT     F333  ; INFRA 4P FRNT#4 PUNCH FWD AL
      MPP
      OUT     T1333 K50
5634  LDFI    F333  ; INFRA 4P FRNT#4 PUNCH FWD AL
      ANI     M4  ; MC RESET SW
      INV
      RST     F333  ; INFRA 4P FRNT#4 PUNCH FWD AL
5641  LD      Y752  ; 4P INFRA WD FRNT#5 HEAD펀치 FWD
      ANI     B524  ; 4P INFRA WELD FRNT#5 PUNCH FWD
      MPS
      AND     T1334
      OUT     F334  ; INFRA 4P FRNT#5 PUNCH FWD AL
      MPP
      OUT     T1334 K50
5652  LDFI    F334  ; INFRA 4P FRNT#5 PUNCH FWD AL
      ANI     M4  ; MC RESET SW
      INV
      RST     F334  ; INFRA 4P FRNT#5 PUNCH FWD AL
5659  LD      Y772  ; 4P INFRA WD REAR#1 HEAD펀치 FWD
      ANI     B530  ; 4P INFRA WELD REAR#1 PUNCH FWD
      MPS
      AND     T1335
      OUT     F335  ; INFRA 4P REAR#1 PUNCH FWD AL
      MPP
      OUT     T1335 K50
5670  LDFI    F335  ; INFRA 4P REAR#1 PUNCH FWD AL
      ANI     M4  ; MC RESET SW
      INV
      RST     F335  ; INFRA 4P REAR#1 PUNCH FWD AL
5677  LD      Y77A  ; 4P INFRA WD REAR#2 HEAD펀치 FWD
      ANI     B531  ; 4P INFRA WELD REAR#2 PUNCH FWD
      MPS
      AND     T1336
      OUT     F336  ; INFRA 4P REAR#2 PUNCH FWD AL
      MPP
      OUT     T1336 K50
5688  LDFI    F336  ; INFRA 4P REAR#2 PUNCH FWD AL
      ANI     M4  ; MC RESET SW
      INV
      RST     F336  ; INFRA 4P REAR#2 PUNCH FWD AL
5695  LD      Y782  ; 4P INFRA WD REAR#3 HEAD펀치 FWD
      ANI     B532  ; 4P INFRA WELD REAR#3 PUNCH FWD
      MPS
      AND     T1337
      OUT     F337  ; INFRA 4P REAR#3 PUNCH FWD AL
      MPP
      OUT     T1337 K50
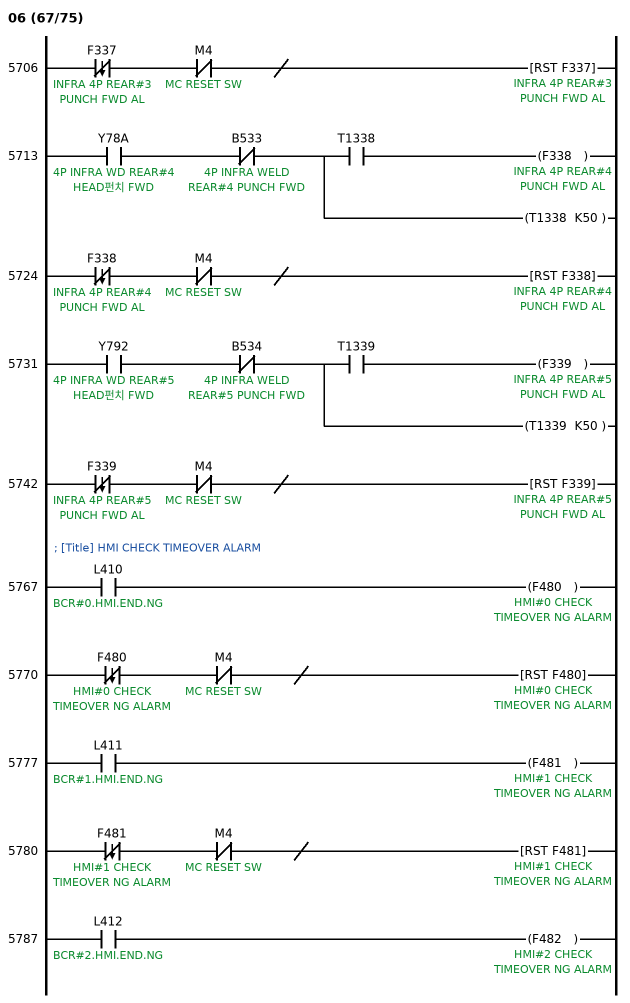
5706  LDFI    F337  ; INFRA 4P REAR#3 PUNCH FWD AL
      ANI     M4  ; MC RESET SW
      INV
      RST     F337  ; INFRA 4P REAR#3 PUNCH FWD AL
5713  LD      Y78A  ; 4P INFRA WD REAR#4 HEAD펀치 FWD
      ANI     B533  ; 4P INFRA WELD REAR#4 PUNCH FWD
      MPS
      AND     T1338
      OUT     F338  ; INFRA 4P REAR#4 PUNCH FWD AL
      MPP
      OUT     T1338 K50
5724  LDFI    F338  ; INFRA 4P REAR#4 PUNCH FWD AL
      ANI     M4  ; MC RESET SW
      INV
      RST     F338  ; INFRA 4P REAR#4 PUNCH FWD AL
5731  LD      Y792  ; 4P INFRA WD REAR#5 HEAD펀치 FWD
      ANI     B534  ; 4P INFRA WELD REAR#5 PUNCH FWD
      MPS
      AND     T1339
      OUT     F339  ; INFRA 4P REAR#5 PUNCH FWD AL
      MPP
      OUT     T1339 K50
5742  LDFI    F339  ; INFRA 4P REAR#5 PUNCH FWD AL
      ANI     M4  ; MC RESET SW
      INV
      RST     F339  ; INFRA 4P REAR#5 PUNCH FWD AL
; [Title] HMI CHECK TIMEOVER ALARM
5767  LD      L410  ; BCR#0.HMI.END.NG
      OUT     F480  ; HMI#0 CHECK TIMEOVER NG ALARM
5770  LDFI    F480  ; HMI#0 CHECK TIMEOVER NG ALARM
      ANI     M4  ; MC RESET SW
      INV
      RST     F480  ; HMI#0 CHECK TIMEOVER NG ALARM
5777  LD      L411  ; BCR#1.HMI.END.NG
      OUT     F481  ; HMI#1 CHECK TIMEOVER NG ALARM
5780  LDFI    F481  ; HMI#1 CHECK TIMEOVER NG ALARM
      ANI     M4  ; MC RESET SW
      INV
      RST     F481  ; HMI#1 CHECK TIMEOVER NG ALARM
5787  LD      L412  ; BCR#2.HMI.END.NG
      OUT     F482  ; HMI#2 CHECK TIMEOVER NG ALARM
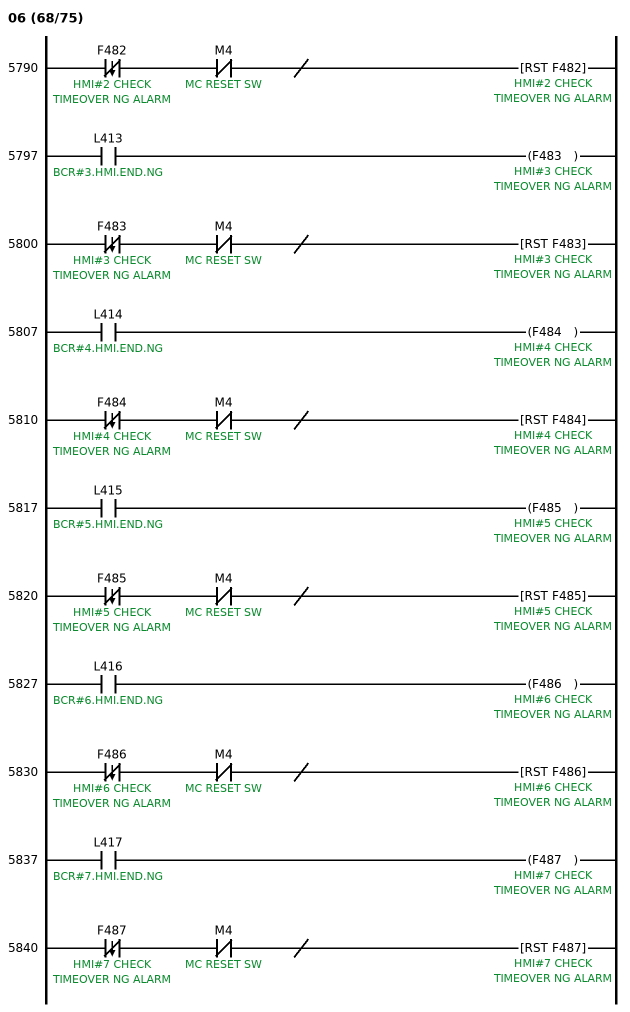
5790  LDFI    F482  ; HMI#2 CHECK TIMEOVER NG ALARM
      ANI     M4  ; MC RESET SW
      INV
      RST     F482  ; HMI#2 CHECK TIMEOVER NG ALARM
5797  LD      L413  ; BCR#3.HMI.END.NG
      OUT     F483  ; HMI#3 CHECK TIMEOVER NG ALARM
5800  LDFI    F483  ; HMI#3 CHECK TIMEOVER NG ALARM
      ANI     M4  ; MC RESET SW
      INV
      RST     F483  ; HMI#3 CHECK TIMEOVER NG ALARM
5807  LD      L414  ; BCR#4.HMI.END.NG
      OUT     F484  ; HMI#4 CHECK TIMEOVER NG ALARM
5810  LDFI    F484  ; HMI#4 CHECK TIMEOVER NG ALARM
      ANI     M4  ; MC RESET SW
      INV
      RST     F484  ; HMI#4 CHECK TIMEOVER NG ALARM
5817  LD      L415  ; BCR#5.HMI.END.NG
      OUT     F485  ; HMI#5 CHECK TIMEOVER NG ALARM
5820  LDFI    F485  ; HMI#5 CHECK TIMEOVER NG ALARM
      ANI     M4  ; MC RESET SW
      INV
      RST     F485  ; HMI#5 CHECK TIMEOVER NG ALARM
5827  LD      L416  ; BCR#6.HMI.END.NG
      OUT     F486  ; HMI#6 CHECK TIMEOVER NG ALARM
5830  LDFI    F486  ; HMI#6 CHECK TIMEOVER NG ALARM
      ANI     M4  ; MC RESET SW
      INV
      RST     F486  ; HMI#6 CHECK TIMEOVER NG ALARM
5837  LD      L417  ; BCR#7.HMI.END.NG
      OUT     F487  ; HMI#7 CHECK TIMEOVER NG ALARM
5840  LDFI    F487  ; HMI#7 CHECK TIMEOVER NG ALARM
      ANI     M4  ; MC RESET SW
      INV
      RST     F487  ; HMI#7 CHECK TIMEOVER NG ALARM
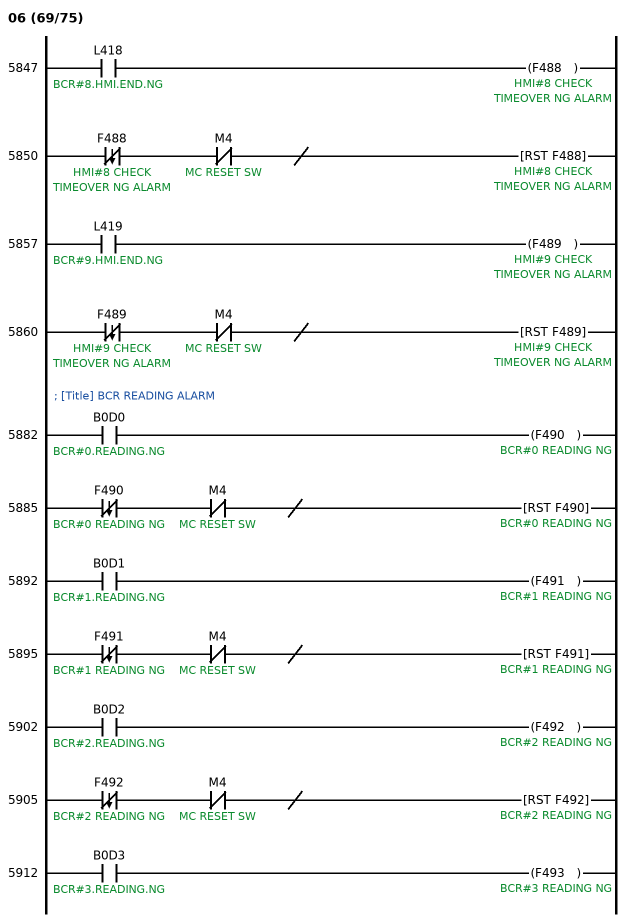
5847  LD      L418  ; BCR#8.HMI.END.NG
      OUT     F488  ; HMI#8 CHECK TIMEOVER NG ALARM
5850  LDFI    F488  ; HMI#8 CHECK TIMEOVER NG ALARM
      ANI     M4  ; MC RESET SW
      INV
      RST     F488  ; HMI#8 CHECK TIMEOVER NG ALARM
5857  LD      L419  ; BCR#9.HMI.END.NG
      OUT     F489  ; HMI#9 CHECK TIMEOVER NG ALARM
5860  LDFI    F489  ; HMI#9 CHECK TIMEOVER NG ALARM
      ANI     M4  ; MC RESET SW
      INV
      RST     F489  ; HMI#9 CHECK TIMEOVER NG ALARM
; [Title] BCR READING ALARM
5882  LD      B0D0  ; BCR#0.READING.NG
      OUT     F490  ; BCR#0 READING NG
5885  LDFI    F490  ; BCR#0 READING NG
      ANI     M4  ; MC RESET SW
      INV
      RST     F490  ; BCR#0 READING NG
5892  LD      B0D1  ; BCR#1.READING.NG
      OUT     F491  ; BCR#1 READING NG
5895  LDFI    F491  ; BCR#1 READING NG
      ANI     M4  ; MC RESET SW
      INV
      RST     F491  ; BCR#1 READING NG
5902  LD      B0D2  ; BCR#2.READING.NG
      OUT     F492  ; BCR#2 READING NG
5905  LDFI    F492  ; BCR#2 READING NG
      ANI     M4  ; MC RESET SW
      INV
      RST     F492  ; BCR#2 READING NG
5912  LD      B0D3  ; BCR#3.READING.NG
      OUT     F493  ; BCR#3 READING NG
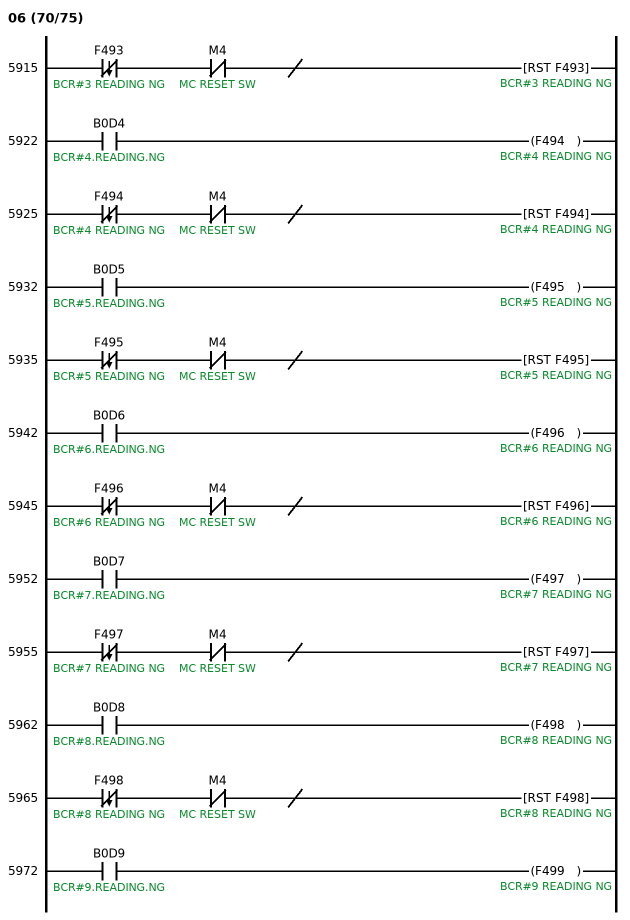
5915  LDFI    F493  ; BCR#3 READING NG
      ANI     M4  ; MC RESET SW
      INV
      RST     F493  ; BCR#3 READING NG
5922  LD      B0D4  ; BCR#4.READING.NG
      OUT     F494  ; BCR#4 READING NG
5925  LDFI    F494  ; BCR#4 READING NG
      ANI     M4  ; MC RESET SW
      INV
      RST     F494  ; BCR#4 READING NG
5932  LD      B0D5  ; BCR#5.READING.NG
      OUT     F495  ; BCR#5 READING NG
5935  LDFI    F495  ; BCR#5 READING NG
      ANI     M4  ; MC RESET SW
      INV
      RST     F495  ; BCR#5 READING NG
5942  LD      B0D6  ; BCR#6.READING.NG
      OUT     F496  ; BCR#6 READING NG
5945  LDFI    F496  ; BCR#6 READING NG
      ANI     M4  ; MC RESET SW
      INV
      RST     F496  ; BCR#6 READING NG
5952  LD      B0D7  ; BCR#7.READING.NG
      OUT     F497  ; BCR#7 READING NG
5955  LDFI    F497  ; BCR#7 READING NG
      ANI     M4  ; MC RESET SW
      INV
      RST     F497  ; BCR#7 READING NG
5962  LD      B0D8  ; BCR#8.READING.NG
      OUT     F498  ; BCR#8 READING NG
5965  LDFI    F498  ; BCR#8 READING NG
      ANI     M4  ; MC RESET SW
      INV
      RST     F498  ; BCR#8 READING NG
5972  LD      B0D9  ; BCR#9.READING.NG
      OUT     F499  ; BCR#9 READING NG
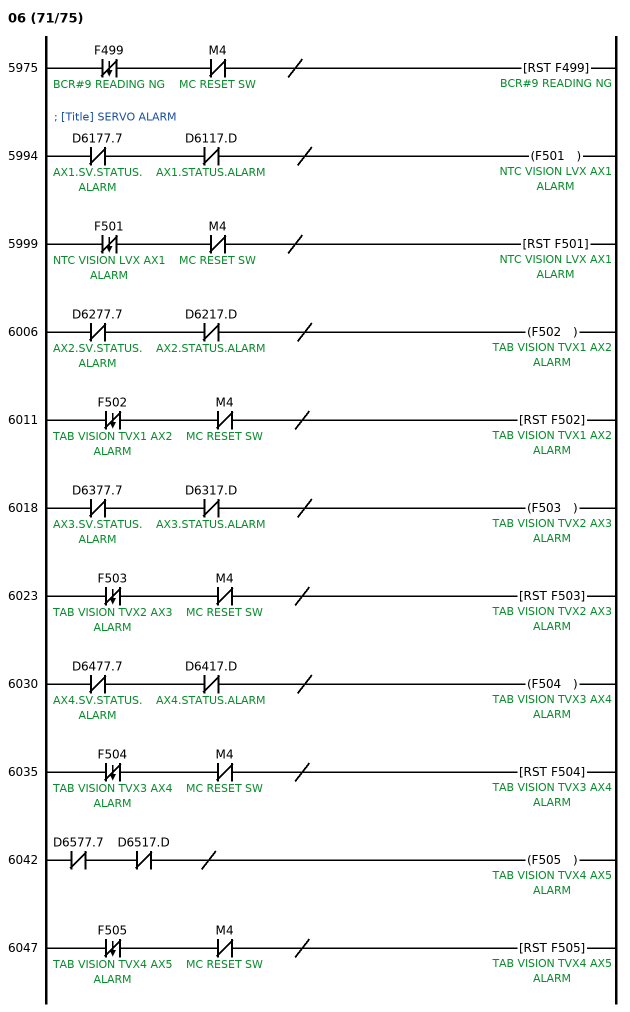
5975  LDFI    F499  ; BCR#9 READING NG
      ANI     M4  ; MC RESET SW
      INV
      RST     F499  ; BCR#9 READING NG
; [Title] SERVO ALARM
5994  LDI     D6177.7  ; AX1.SV.STATUS.ALARM
      ANI     D6117.D  ; AX1.STATUS.ALARM
      INV
      OUT     F501  ; NTC VISION LVX AX1 ALARM
5999  LDFI    F501  ; NTC VISION LVX AX1 ALARM
      ANI     M4  ; MC RESET SW
      INV
      RST     F501  ; NTC VISION LVX AX1 ALARM
6006  LDI     D6277.7  ; AX2.SV.STATUS.ALARM
      ANI     D6217.D  ; AX2.STATUS.ALARM
      INV
      OUT     F502  ; TAB VISION TVX1 AX2 ALARM
6011  LDFI    F502  ; TAB VISION TVX1 AX2 ALARM
      ANI     M4  ; MC RESET SW
      INV
      RST     F502  ; TAB VISION TVX1 AX2 ALARM
6018  LDI     D6377.7  ; AX3.SV.STATUS.ALARM
      ANI     D6317.D  ; AX3.STATUS.ALARM
      INV
      OUT     F503  ; TAB VISION TVX2 AX3 ALARM
6023  LDFI    F503  ; TAB VISION TVX2 AX3 ALARM
      ANI     M4  ; MC RESET SW
      INV
      RST     F503  ; TAB VISION TVX2 AX3 ALARM
6030  LDI     D6477.7  ; AX4.SV.STATUS.ALARM
      ANI     D6417.D  ; AX4.STATUS.ALARM
      INV
      OUT     F504  ; TAB VISION TVX3 AX4 ALARM
6035  LDFI    F504  ; TAB VISION TVX3 AX4 ALARM
      ANI     M4  ; MC RESET SW
      INV
      RST     F504  ; TAB VISION TVX3 AX4 ALARM
6042  LDI     D6577.7
      ANI     D6517.D
      INV
      OUT     F505  ; TAB VISION TVX4 AX5 ALARM
6047  LDFI    F505  ; TAB VISION TVX4 AX5 ALARM
      ANI     M4  ; MC RESET SW
      INV
      RST     F505  ; TAB VISION TVX4 AX5 ALARM
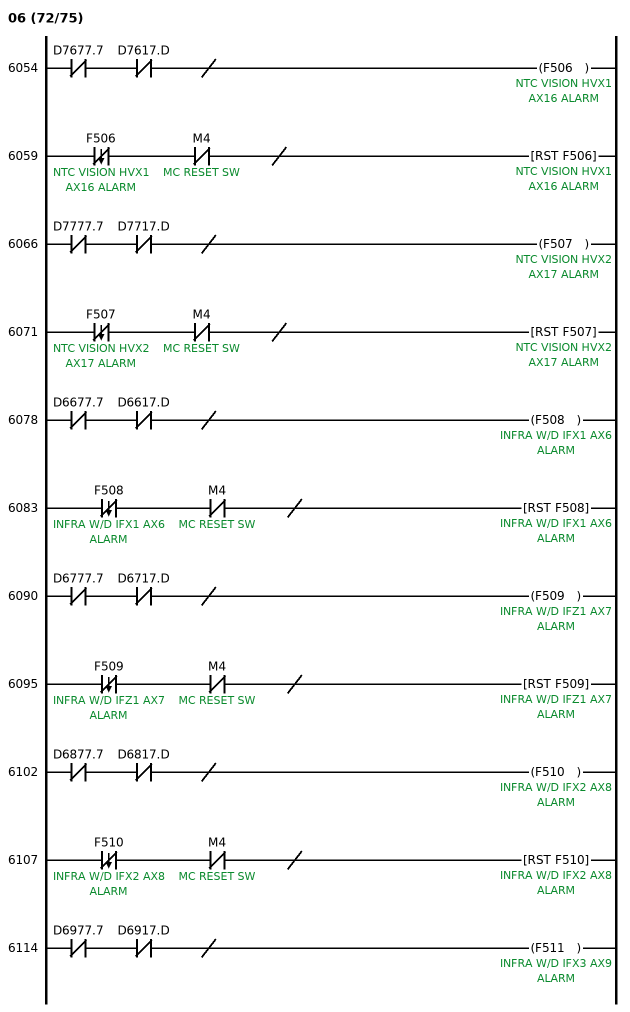
6054  LDI     D7677.7
      ANI     D7617.D
      INV
      OUT     F506  ; NTC VISION HVX1 AX16 ALARM
6059  LDFI    F506  ; NTC VISION HVX1 AX16 ALARM
      ANI     M4  ; MC RESET SW
      INV
      RST     F506  ; NTC VISION HVX1 AX16 ALARM
6066  LDI     D7777.7
      ANI     D7717.D
      INV
      OUT     F507  ; NTC VISION HVX2 AX17 ALARM
6071  LDFI    F507  ; NTC VISION HVX2 AX17 ALARM
      ANI     M4  ; MC RESET SW
      INV
      RST     F507  ; NTC VISION HVX2 AX17 ALARM
6078  LDI     D6677.7
      ANI     D6617.D
      INV
      OUT     F508  ; INFRA W/D IFX1 AX6 ALARM
6083  LDFI    F508  ; INFRA W/D IFX1 AX6 ALARM
      ANI     M4  ; MC RESET SW
      INV
      RST     F508  ; INFRA W/D IFX1 AX6 ALARM
6090  LDI     D6777.7
      ANI     D6717.D
      INV
      OUT     F509  ; INFRA W/D IFZ1 AX7 ALARM
6095  LDFI    F509  ; INFRA W/D IFZ1 AX7 ALARM
      ANI     M4  ; MC RESET SW
      INV
      RST     F509  ; INFRA W/D IFZ1 AX7 ALARM
6102  LDI     D6877.7
      ANI     D6817.D
      INV
      OUT     F510  ; INFRA W/D IFX2 AX8 ALARM
6107  LDFI    F510  ; INFRA W/D IFX2 AX8 ALARM
      ANI     M4  ; MC RESET SW
      INV
      RST     F510  ; INFRA W/D IFX2 AX8 ALARM
6114  LDI     D6977.7
      ANI     D6917.D
      INV
      OUT     F511  ; INFRA W/D IFX3 AX9 ALARM
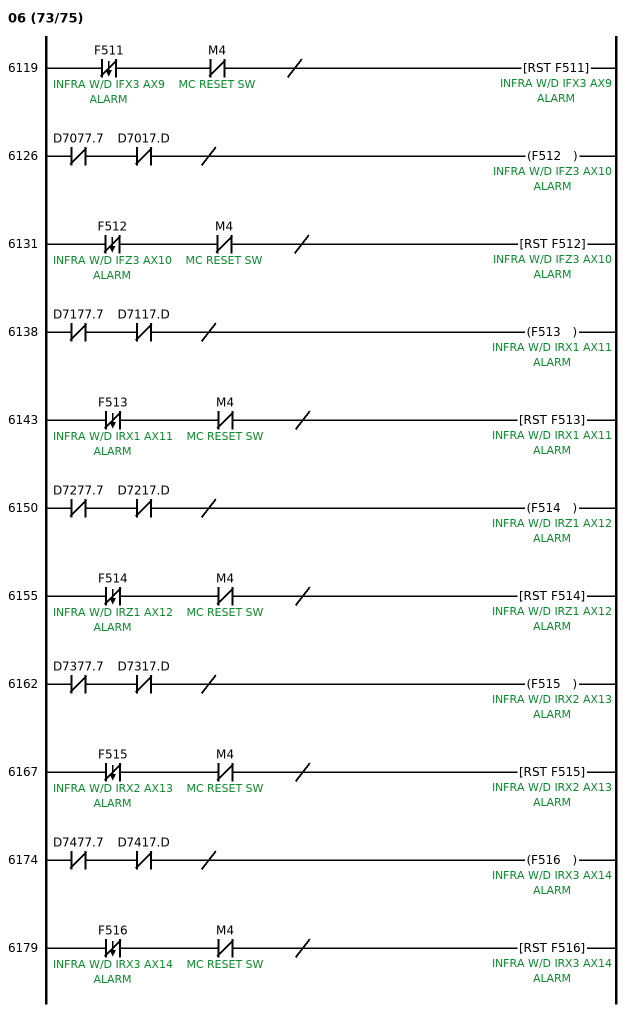
6119  LDFI    F511  ; INFRA W/D IFX3 AX9 ALARM
      ANI     M4  ; MC RESET SW
      INV
      RST     F511  ; INFRA W/D IFX3 AX9 ALARM
6126  LDI     D7077.7
      ANI     D7017.D
      INV
      OUT     F512  ; INFRA W/D IFZ3 AX10 ALARM
6131  LDFI    F512  ; INFRA W/D IFZ3 AX10 ALARM
      ANI     M4  ; MC RESET SW
      INV
      RST     F512  ; INFRA W/D IFZ3 AX10 ALARM
6138  LDI     D7177.7
      ANI     D7117.D
      INV
      OUT     F513  ; INFRA W/D IRX1 AX11 ALARM
6143  LDFI    F513  ; INFRA W/D IRX1 AX11 ALARM
      ANI     M4  ; MC RESET SW
      INV
      RST     F513  ; INFRA W/D IRX1 AX11 ALARM
6150  LDI     D7277.7
      ANI     D7217.D
      INV
      OUT     F514  ; INFRA W/D IRZ1 AX12 ALARM
6155  LDFI    F514  ; INFRA W/D IRZ1 AX12 ALARM
      ANI     M4  ; MC RESET SW
      INV
      RST     F514  ; INFRA W/D IRZ1 AX12 ALARM
6162  LDI     D7377.7
      ANI     D7317.D
      INV
      OUT     F515  ; INFRA W/D IRX2 AX13 ALARM
6167  LDFI    F515  ; INFRA W/D IRX2 AX13 ALARM
      ANI     M4  ; MC RESET SW
      INV
      RST     F515  ; INFRA W/D IRX2 AX13 ALARM
6174  LDI     D7477.7
      ANI     D7417.D
      INV
      OUT     F516  ; INFRA W/D IRX3 AX14 ALARM
6179  LDFI    F516  ; INFRA W/D IRX3 AX14 ALARM
      ANI     M4  ; MC RESET SW
      INV
      RST     F516  ; INFRA W/D IRX3 AX14 ALARM
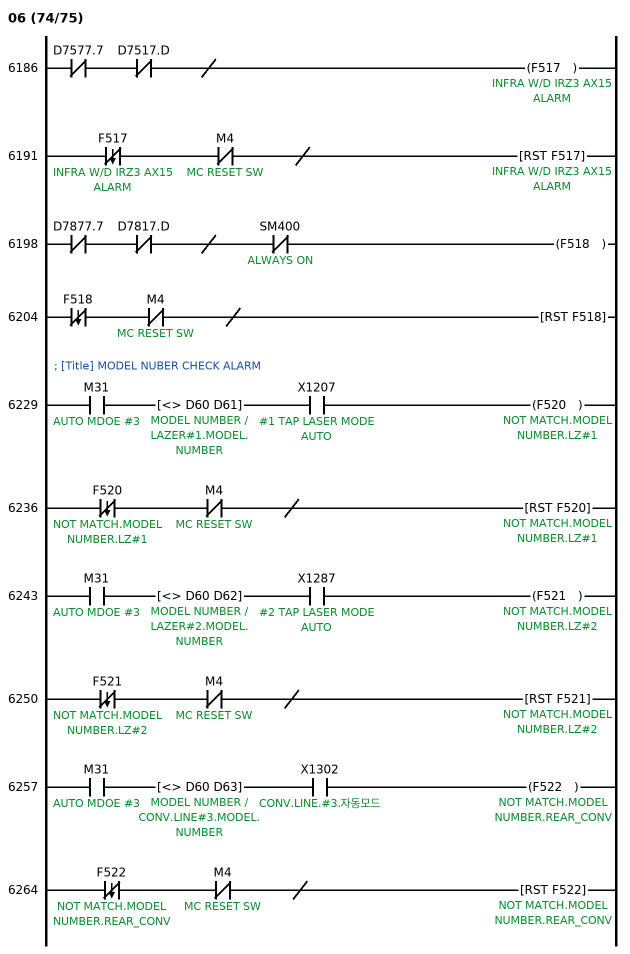
6186  LDI     D7577.7
      ANI     D7517.D
      INV
      OUT     F517  ; INFRA W/D IRZ3 AX15 ALARM
6191  LDFI    F517  ; INFRA W/D IRZ3 AX15 ALARM
      ANI     M4  ; MC RESET SW
      INV
      RST     F517  ; INFRA W/D IRZ3 AX15 ALARM
6198  LDI     D7877.7
      ANI     D7817.D
      INV
      ANI     SM400  ; ALWAYS ON
      OUT     F518
6204  LDFI    F518
      ANI     M4  ; MC RESET SW
      INV
      RST     F518
; [Title] MODEL NUBER CHECK ALARM
6229  LD      M31  ; AUTO MDOE #3
      AND<>   D60 D61  ; MODEL NUMBER / LAZER#1.MODEL.NUMBER
      AND     X1207  ; #1 TAP LASER MODE AUTO
      OUT     F520  ; NOT MATCH.MODEL NUMBER.LZ#1
6236  LDFI    F520  ; NOT MATCH.MODEL NUMBER.LZ#1
      ANI     M4  ; MC RESET SW
      INV
      RST     F520  ; NOT MATCH.MODEL NUMBER.LZ#1
6243  LD      M31  ; AUTO MDOE #3
      AND<>   D60 D62  ; MODEL NUMBER / LAZER#2.MODEL.NUMBER
      AND     X1287  ; #2 TAP LASER MODE AUTO
      OUT     F521  ; NOT MATCH.MODEL NUMBER.LZ#2
6250  LDFI    F521  ; NOT MATCH.MODEL NUMBER.LZ#2
      ANI     M4  ; MC RESET SW
      INV
      RST     F521  ; NOT MATCH.MODEL NUMBER.LZ#2
6257  LD      M31  ; AUTO MDOE #3
      AND<>   D60 D63  ; MODEL NUMBER / CONV.LINE#3.MODEL.NUMBER
      AND     X1302  ; CONV.LINE.#3.자동모드
      OUT     F522  ; NOT MATCH.MODEL NUMBER.REAR_CONV
6264  LDFI    F522  ; NOT MATCH.MODEL NUMBER.REAR_CONV
      ANI     M4  ; MC RESET SW
      INV
      RST     F522  ; NOT MATCH.MODEL NUMBER.REAR_CONV
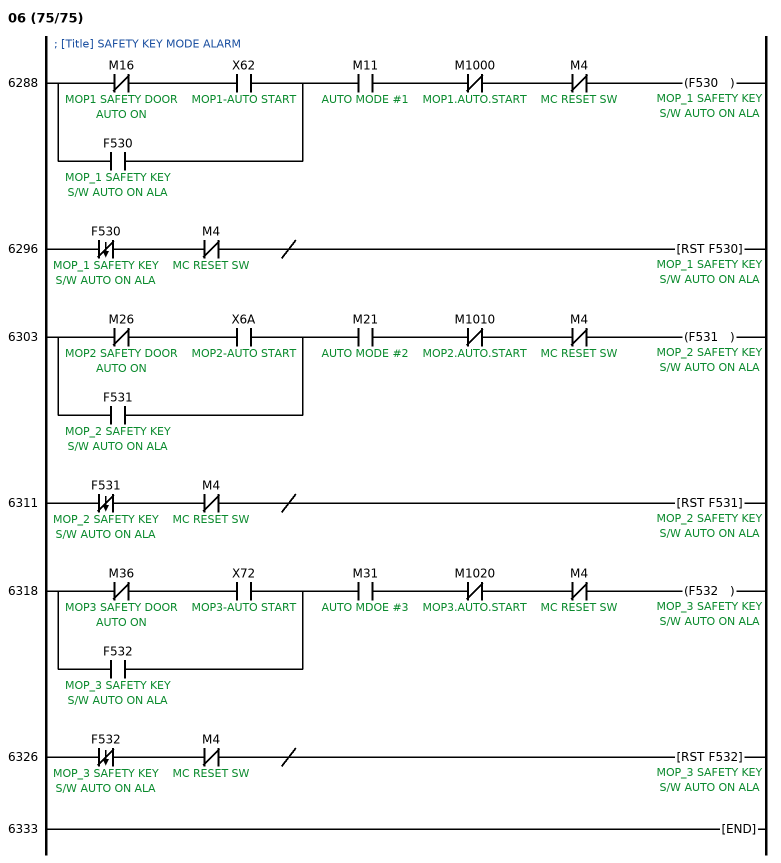
; [Title] SAFETY KEY MODE ALARM
6288  LDI     M16  ; MOP1 SAFETY DOOR AUTO ON
      AND     X62  ; MOP1-AUTO START
      OR      F530  ; MOP_1 SAFETY KEY S/W AUTO ON ALA
      AND     M11  ; AUTO MODE #1
      ANI     M1000  ; MOP1.AUTO.START
      ANI     M4  ; MC RESET SW
      OUT     F530  ; MOP_1 SAFETY KEY S/W AUTO ON ALA
6296  LDFI    F530  ; MOP_1 SAFETY KEY S/W AUTO ON ALA
      ANI     M4  ; MC RESET SW
      INV
      RST     F530  ; MOP_1 SAFETY KEY S/W AUTO ON ALA
6303  LDI     M26  ; MOP2 SAFETY DOOR AUTO ON
      AND     X6A  ; MOP2-AUTO START
      OR      F531  ; MOP_2 SAFETY KEY S/W AUTO ON ALA
      AND     M21  ; AUTO MODE #2
      ANI     M1010  ; MOP2.AUTO.START
      ANI     M4  ; MC RESET SW
      OUT     F531  ; MOP_2 SAFETY KEY S/W AUTO ON ALA
6311  LDFI    F531  ; MOP_2 SAFETY KEY S/W AUTO ON ALA
      ANI     M4  ; MC RESET SW
      INV
      RST     F531  ; MOP_2 SAFETY KEY S/W AUTO ON ALA
6318  LDI     M36  ; MOP3 SAFETY DOOR AUTO ON
      AND     X72  ; MOP3-AUTO START
      OR      F532  ; MOP_3 SAFETY KEY S/W AUTO ON ALA
      AND     M31  ; AUTO MDOE #3
      ANI     M1020  ; MOP3.AUTO.START
      ANI     M4  ; MC RESET SW
      OUT     F532  ; MOP_3 SAFETY KEY S/W AUTO ON ALA
6326  LDFI    F532  ; MOP_3 SAFETY KEY S/W AUTO ON ALA
      ANI     M4  ; MC RESET SW
      INV
      RST     F532  ; MOP_3 SAFETY KEY S/W AUTO ON ALA
6333  END
END_PROGRAM

// device comments not shown above
X17  ; 0000:Axis 8 BUSY
X18  ; 0000:Axis 9  BUSY
X19  ; 0000:Axis 10  BUSY
X1A  ; 0000:Axis 11  BUSY
X1B  ; 0000:Axis 12 BUSY
X1C  ; 0000:Axis 13  BUSY
X1D  ; 0000:Axis 14  BUSY
X1E  ; 0000:Axis 15  BUSY
X1F  ; 0000:Axis 16 BUSY
X3A  ; 0000:Axis 11  BUSY
X3B  ; 0000:Axis 12 BUSY
X3C  ; 0000:Axis 13  BUSY
X3D  ; 0000:Axis 14  BUSY
X3E  ; 0000:Axis 15  BUSY
X3F  ; 0000:Axis 16 BUSY
X831  ; 트리거 실패
X871  ; 코맨드명령실행 완료 (핸드쉐이크)
X872  ; 코맨드명령실행 에러 (핸드쉐이크)
X873  ; 일치도 갱신 잠금상태
X88F  ; 프로그램 전환 실패
X8B1  ; 트리거 실패
X8F1  ; 코맨드명령실행 완료 (핸드쉐이크)
X8F2  ; 코맨드명령실행 에러 (핸드쉐이크)
X8F3  ; 일치도 갱신 잠금상태
X90F  ; 프로그램 전환 실패
X1305  ; MODEL BIT #2
X1306  ; MODEL BIT #3
X1307  ; MODEL BIT #4
Y17  ; 0000:Axis 8 Positioning start
Y18  ; 0000:Axis 9  Positioning  start
Y19  ; 0000:Axis 10  Positioning  start
Y1A  ; 0000:Axis 11 Positioning start
Y1B  ; 0000:Axis 12 Positioning start
Y1C  ; 0000:Axis 13  Positioning  start
Y1D  ; 0000:Axis 14  Positioning  start
Y1E  ; 0000:Axis 15 Positioning start
Y1F  ; 0000:Axis 16 Positioning start
Y3A  ; 0020:Axis 11 Positioning start
Y3B  ; 0020:Axis 12 Positioning start
Y3C  ; 0020:Axis 13  Positioning  start
Y3D  ; 0020:Axis 14  Positioning  start
Y3E  ; 0020:Axis 15 Positioning start
Y3F  ; 0020:Axis 16 Positioning start
Y1305  ; MODEL BIT #2
Y1306  ; MODEL BIT #3
Y1307  ; MODEL BIT #4
M200  ; MANUAL FWD CMD
M300  ; MANUAL BWD CMD
M400  ; MANU 1 FWD
M500  ; MANU 1 BWD
M1114  ; AX1.SERVO.OFF
M1118  ; AX1.SV.ON.상태
M1124  ; AX2.SERVO.OFF
M1128  ; AX2.SV.ON.상태
M1134  ; AX3.SERVO.OFF
M1138  ; AX3.SV.ON.상태
M1144  ; AX4.SERVO.OFF
M1154  ; AX5.SERVO.OFF
M1164  ; AX6.SERVO.OFF
M1174  ; AX7.SERVO.OFF
M1184  ; AX8.SERVO.OFF
M1194  ; AX9.SERVO.OFF
M1204  ; AX10.SERVO.OFF
M1214  ; AX11.SERVO.OFF
M1224  ; AX12.SERVO.OFF
M1234  ; AX13.SERVO.OFF
M1244  ; AX14.SERVO.OFF
M1254  ; AX15.SERVO.OFF
M1264  ; AX16.SERVO.OFF
M1274  ; AX17.SERVO.OFF
M4000  ; 컨베어 투입부 자동 사이클
D350  ; TH.VISION.COUNTER
D352  ; TH.VISION.COUNTER
D382  ; MOP2 SECURITY LEVEL
D812  ; AX1. ACC TIME
D814  ; AX1.DEC TIME
D822  ; AX2. ACC TIME
D824  ; AX2.DEC TIME
D832  ; AX3. ACC TIME
D834  ; AX3.DEC TIME
D842  ; AX4. ACC TIME
D844  ; AX4.DEC TIME
D852  ; AX5. ACC TIME
D854  ; AX5.DEC TIME
D862  ; AX6. ACC TIME
D864  ; AX6.DEC TIME
D872  ; AX7. ACC TIME
D874  ; AX7.DEC TIME
D882  ; AX8. ACC TIME
D884  ; AX8.DEC TIME
D892  ; AX9. ACC TIME
D894  ; AX9.DEC TIME
D902  ; AX10. ACC TIME
D904  ; AX10.DEC TIME
D912  ; AX11. ACC TIME
D914  ; AX11.DEC TIME
D922  ; AX12. ACC TIME
D924  ; AX12.DEC TIME
D932  ; AX13. ACC TIME
D934  ; AX13.DEC TIME
D942  ; AX14. ACC TIME
D944  ; AX14.DEC TIME
D952  ; AX15. ACC TIME
D954  ; AX15.DEC TIME
D962  ; AX16. ACC TIME
D964  ; AX16.DEC TIME
D972  ; AX17. ACC TIME
D974  ; AX17.DEC TIME
D980  ; AX18. JOG SPEED
D982  ; AX18. ACC TIME
D984  ; AX18.DEC TIME
D990  ; AX19. JOG SPEED
D992  ; AX19. ACC TIME
D994  ; AX19.DEC TIME
D1001  ; AX1
D1003  ; AX1
D1005  ; AX2
D1007  ; AX2
D1009  ; AX3
D1011  ; AX3
D1013  ; AX4
D1015  ; AX4
D1017  ; AX5
D1019  ; AX5
D1021  ; AX6
D1023  ; AX6
D1025  ; AX7
D1027  ; AX7
D1029  ; AX8
D1031  ; AX8
D1033  ; AX9
D1035  ; AX9
D1037  ; AX10
D1039  ; AX10
D1041  ; AX11
D1043  ; AX11
D1045  ; AX12
D1047  ; AX12
D1049  ; AX13
D1051  ; AX13
D1053  ; AX14
D1055  ; AX14
D1057  ; AX15
D1059  ; AX15
D1061  ; AX16
D1063  ; AX16
D1065  ; AX17
D1067  ; AX17
D5600  ; 비젼2.출력완료
D5601  ; 비젼2.출력제어
D5610  ; 비젼2.출력결과
D6106  ; AX1.ERROR.NUM
D6117  ; AX1.STATUS
D6177  ; AX1.SV.STATUS
D6179  ; AX1.LOAD
D6206  ; AX2.ERROR.NUM
D6217  ; AX2.STATUS
D6277  ; AX2.SV.STATUS
D6279  ; AX2.LOAD
D6306  ; AX3.ERROR.NUM
D6317  ; AX3.STATUS
D6377  ; AX3.SV.STATUS
D6379  ; AX3.LOAD
D6406  ; AX4.ERROR.NUM
D6417  ; AX4.STATUS
D6477  ; AX4.SV.STATUS
D6479  ; AX4.LOAD
D6506  ; AX5.ERROR.NUM
D6517  ; AX5.STATUS
D6577  ; AX5.SV.STATUS
D6579  ; AX5.LOAD
D6606  ; AX6.ERROR.NUM
D6617  ; AX6.STATUS
D6677  ; AX6.SV.STATUS
D6679  ; AX6.LOAD
D6706  ; AX7.ERROR.NUM
D6717  ; AX7.STATUS
D6777  ; AX7.SV.STATUS
D6779  ; AX7.LOAD
D6806  ; AX8.ERROR.NUM
D6817  ; AX8.STATUS
D6877  ; AX8.SV.STATUS
D6879  ; AX8.LOAD
D6906  ; AX9.ERROR.NUM
D6917  ; AX9.STATUS
D6977  ; AX9.SV.STATUS
D6979  ; AX9.LOAD
D7006  ; AX10.ERROR.NUM
D7017  ; AX10.STATUS
D7077  ; AX10.SV.STATUS
D7079  ; AX10.LOAD
D7106  ; AX11.ERROR.NUM
D7117  ; AX11.STATUS
D7177  ; AX11.SV.STATUS
D7179  ; AX11.LOAD
D7206  ; AX12.ERROR.NUM
D7217  ; AX12.STATUS
D7277  ; AX12.SV.STATUS
D7279  ; AX12.LOAD
D7306  ; AX13.ERROR.NUM
D7317  ; AX13.STATUS
D7377  ; AX13.SV.STATUS
D7379  ; AX13.LOAD
D7406  ; AX14.ERROR.NUM
D7417  ; AX14.STATUS
D7477  ; AX14.SV.STATUS
D7479  ; AX14.LOAD
D7506  ; AX15.ERROR.NUM
D7517  ; AX15.STATUS
D7577  ; AX15.SV.STATUS
D7579  ; AX15.LOAD
D7606  ; AX16.ERROR.NUM
D7617  ; AX16.STATUS
D7677  ; AX16.SV.STATUS
D7679  ; AX16.LOAD
D7706  ; AX17.ERROR.NUM
D7717  ; AX17.STATUS
D7777  ; AX17.SV.STATUS
D7779  ; AX17.LOAD
D7800  ; AX18.FEED.VALUE
D7806  ; AX18.ERROR.NUM
D7817  ; AX18.STATUS
D7877  ; AX18.SV.STATUS
D7879  ; AX18.LOAD
B8D  ; 임시.비젼.이동명령6
B1114  ; AX1.위치4
B1115  ; AX1.위치5
B1116  ; AX1.위치6
B1124  ; AX2.위치4
B1125  ; AX2.위치5
B1126  ; AX2.위치6
B1134  ; AX3.위치4
B1135  ; AX3.위치5
B1136  ; AX3.위치6
B1144  ; AX4.위치4
B1145  ; AX4.위치5
B1146  ; AX4.위치6
B1154  ; AX5.위치4
B1155  ; AX5.위치5
B1156  ; AX5.위치6
B1212  ; AX6.위치2
B1213  ; AX6.위치3
B1214  ; AX6.위치4
B1215  ; AX6.위치5
B1216  ; AX6.위치6
B1222  ; AX7.위치2
B1223  ; AX7.위치3
B1224  ; AX7.위치4
B1225  ; AX7.위치5
B1226  ; AX7.위치6
B1232  ; AX8.위치2
B1233  ; AX8.위치3
B1234  ; AX8.위치4
B1235  ; AX8.위치5
B1236  ; AX8.위치6
B1242  ; AX9.위치2
B1243  ; AX9.위치3
B1244  ; AX9.위치4
B1245  ; AX9.위치5
B1246  ; AX9.위치6
B1252  ; AX10.위치2
B1253  ; AX10.위치3
B1254  ; AX10.위치4
B1255  ; AX10.위치5
B1256  ; AX10.위치6
B1262  ; AX11.위치2
B1263  ; AX11.위치3
B1264  ; AX11.위치4
B1265  ; AX11.위치5
B1266  ; AX11.위치6
B1272  ; AX12.위치2
B1273  ; AX12.위치3
B1274  ; AX12.위치4
B1275  ; AX12.위치5
B1276  ; AX12.위치6
B1282  ; AX13.위치2
B1283  ; AX13.위치3
B1284  ; AX13.위치4
B1285  ; AX13.위치5
B1286  ; AX13.위치6
B1292  ; AX14.위치2
B1293  ; AX14.위치3
B1294  ; AX14.위치4
B1295  ; AX14.위치5
B1296  ; AX14.위치6
B12A2  ; AX15.위치2
B12A3  ; AX15.위치3
B12A4  ; AX15.위치4
B12A5  ; AX15.위치5
B12A6  ; AX15.위치6
B12B4  ; AX16.위치4
B12B5  ; AX16.위치5
B12B6  ; AX16.위치6
B12C4  ; AX17.위치4
B12C5  ; AX17.위치5
B12C6  ; AX17.위치6
L120  ; 2P INFRA WELDING REAR END
L140  ; 4P INFRA WELDING REAR END
L207  ; VISION.1-7.OK
L208  ; VISION.1-8.OK
L209  ; VISION.1-9.OK
L217  ; VISION.1-7.NG
L218  ; VISION.1-8.NG
L219  ; VISION.1-9.NG
L227  ; VISION.2-7.OK
L228  ; VISION.2-8.OK
L229  ; VISION.2-9.OK
L237  ; VISION.2-7.NG
L238  ; VISION.2-8.NG
L239  ; VISION.2-9.NG
F1001  ; VISION  PALLET POS` UP/DN ALARM
F1002  ; EOL 2P PALLET POS` UP/DN ALARM
F1003  ; EOL 4P PALLET POS` UP/DN ALARM
F1004  ; LABEL BARCODE PALLET POS UP/DN A
F1005  ; NG 배출 UNIT DIVERTER UP/DN ALAR
F1007  ; WORK UNLOAD POS` PALLET CLAMP/UN
F1008  ; WORK UNLOAD POS`PALLET탈착UP/DN1
F1009  ; WORK UNLOAD POS`PALLET탈착UP/DN2
F1011  ; OUT CON`V LIFT  UP/DN ALARM
F1012  ; MAIN 상부 CON`V  CHAIN CHECK ALA
F1013  ; MAIN 하부 CON`V  CHAIN CHECK ALA
F1014  ; CLAMP UNIT (2P-18S) UP/DN ALARM
F1015  ; CONNECT CLAMP(2P-18S) CLAMP/UNCL
F1016  ; CONNECTOR CLAMP(2P-18S) FWD/BWD
F1017  ; BUS BAR CLEANING(FRONT) UP/DN AL
F1018  ; BUS BAR CLEANING(REAR) UP/DN ALA
F1019  ; EOL_PIN CHECK(2P-18S-S) FWD/BWD
F1020  ; EOL_PIN CHECK(2P-18S-R) FWD/BWD
F1021  ; BUSBAR CHECK #1(FRONT)FWD/BWD_2P
F1022  ; BUSBAR CHECK #2(FRONT)FWD/BWD_2P
F1023  ; BUSBAR CHECK #3(FRONT)FWD/BWD_2P
F1024  ; BUSBAR CHECK #4(FRONT)FWD/BWD_2P
F1025  ; BUSBAR CHECK #5(FRONT)FWD/BWD_2P
F1026  ; BUSBAR CHECK #6(FRONT)FWD/BWD_2P
F1027  ; BUSBAR CHECK #7(FRONT)FWD/BWD_2P
F1028  ; BUSBAR CHECK #8(FRONT)FWD/BWD_2P
F1029  ; BUSBAR CHECK #9(FRONT)FWD/BWD_2P
F1030  ; BUSBAR CHECK#10(FRONT)FWD/BWD_2P
F1031  ; BUSBAR CHECK #1(REAR)FWD/BWD_2P
F1032  ; BUSBAR CHECK #2(REAR)FWD/BWD_2P
F1033  ; BUSBAR CHECK #3(REAR)FWD/BWD_2P
F1034  ; BUSBAR CHECK #4(REAR)FWD/BWD_2P
F1035  ; BUSBAR CHECK #5(REAR)FWD/BWD_2P
F1036  ; BUSBAR CHECK #6(REAR)FWD/BWD_2P
F1037  ; BUSBAR CHECK #7(REAR)FWD/BWD_2P
F1038  ; BUSBAR CHECK #8(REAR)FWD/BWD_2P
F1039  ; BUSBAR CHECK #9(REAR)FWD/BWD_2P
F1040  ; CLAMP UNIT (4P-8S) UP/DN ALARM
F1041  ; CONNECTOR CLAMP(4P-8S) CLAMP/UNC
F1042  ; CONNECTOR CLAMP(4P-8S) FWD/BWD
F1043  ; CLAMP UNIT (4P-10S) UP/DOWN ALAR
F1044  ; CONNECTOR CLAMP(4P-10S) CLAMP/UN
F1045  ; CONNECTOR CLAMP(4P-10S) FWD/BWD
F1046  ; CONNECTOR CLAMP(4P-10S-S) FWD/BW
F1047  ; CONNECTOR CLAMP(4P-10S-R) FWD/BW
F1048  ; BUS BAR CLEANING(FRONT) UP/DN AL
F1049  ; BUS BAR CLEANING(REAR) UP/DN ALA
F1131  ; EOL_CLAMP   UNIT(2P-18S) UP ALAR
F1132  ; CLAMP UNIT (2P-18S) DOWN ALARM
F1133  ; EOL_CONNECT CLAMP(2P-18S)CLAMP A
F1134  ; EOL_CONNECT CLAMP(2P-18S)UNCLAMP
F1135  ; EOL_CONNECT CLAMP(2P-18S) FWD AL
F1136  ; EOL_CONNECT CLAMP(2P-18S) BWD AL
F1137  ; EOL_BUS BAR CLEAN(FRONT) UP ALAR
F1138  ; EOL_BUS BAR CLEAN(FRONT) DOWN AL
F1139  ; EOL_BUS BAR CLEAN(REAR) UP ALARM
F1140  ; EOL_BUS BAR CLEAN(REAR) DOWN ALA
F1141  ; EOL_PIN CHECK(2P-18S-S) FWD ALAR
F1142  ; EOL_PIN CHECK(2P-18S-S) BWD ALAR
F1143  ; EOL_PIN CHECK(2P-18S-R) FWD ALAR
F1144  ; EOL_PIN CHECK(2P-18S-R) BWD ALAR
F1150  ; BUSBAR CHECK#1(FRONT)FWD_2P ALA
F1151  ; BUSBAR CHECK#1(FRONT)BWD_2P ALA
F1152  ; BUSBAR CHECK#2(FRONT)FWD_2P ALA
F1153  ; BUSBAR CHECK#2(FRONT)BWD_2P ALA
F1154  ; BUSBAR CHECK#3(FRONT)FWD_2P ALA
F1155  ; BUSBAR CHECK#3(FRONT)BWD_2P ALA
F1156  ; BUSBAR CHECK#4(FRONT)FWD_2P ALA
F1157  ; BUSBAR CHECK#4(FRONT)BWD_2P ALA
F1158  ; BUSBAR CHECK#5(FRONT)FWD_2P ALA
F1159  ; BUSBAR CHECK#5(FRONT)BWD_2P ALA
F1160  ; BUSBAR CHECK#6(FRONT)FWD_2P ALA
F1161  ; BUSBAR CHECK#6(FRONT)BWD_2P ALA
F1162  ; BUSBAR CHECK#7(FRONT)FWD_2P ALA
F1163  ; BUSBAR CHECK#7(FRONT)BWD_2P ALA
F1164  ; BUSBAR CHECK#8(FRONT)FWD_2P ALA
F1165  ; BUSBAR CHECK#8(FRONT)BWD_2P ALA
F1166  ; BUSBAR CHECK#9(FRONT)FWD_2P ALA
F1167  ; BUSBAR CHECK#9(FRONT)BWD_2P ALA
F1168  ; BUSBAR CHECK#10(FRONT)FWD_2P ALA
F1169  ; BUSBAR CHECK#10(FRONT)BWD_2P ALA
F1170  ; BUSBAR CHECK#1(REAR)FWD_2P ALA
F1171  ; BUSBAR CHECK#1(REAR)BWD_2P ALA
F1172  ; BUSBAR CHECK#2(REAR)FWD_2P ALA
F1173  ; BUSBAR CHECK#2(REAR)BWD_2P ALA
F1174  ; BUSBAR CHECK#3(REAR)FWD_2P ALA
F1175  ; BUSBAR CHECK#3(REAR)BWD_2P ALA
F1176  ; BUSBAR CHECK#4(REAR)FWD_2P ALA
F1177  ; BUSBAR CHECK#4(REAR)BWD_2P ALA
F1178  ; BUSBAR CHECK#5(REAR)FWD_2P ALA
F1179  ; BUSBAR CHECK#5(REAR)BWD_2P ALA
F1180  ; BUSBAR CHECK#6(REAR)FWD_2P ALA
F1181  ; BUSBAR CHECK#6(REAR)BWD_2P ALA
F1182  ; BUSBAR CHECK#7(REAR)FWD_2P ALA
F1183  ; BUSBAR CHECK#7(REAR)BWD_2P ALA
F1184  ; BUSBAR CHECK#8(REAR)FWD_2P ALA
F1185  ; BUSBAR CHECK#8(REAR)BWD_2P ALA
F1186  ; BUSBAR CHECK#9(REAR)FWD_2P ALA
F1187  ; BUSBAR CHECK#9(REAR)BWD_2P ALA
F1190  ; CLAMP UNIT (4P-8S) UP ALARM
F1191  ; CLAMP UNIT (4P-8S) DOWN ALARM
F1192  ; CONNECTOR CLAMP(4P-8S) CLAMP ALA
F1193  ; CONNECTOR CLAMP(4P-8S) UNCLAMP A
F1194  ; CONNECTOR CLAMP(4P-8S) FWD ALARM
F1195  ; CONNECTOR CLAMP(4P-8S) BWD ALARM
F1196  ; CLAMP UNIT (4P-10S) UP ALARM
F1197  ; CLAMP UNIT (4P-10S) DOWN ALARM
F1198  ; CONNECTOR CLAMP(4P-10S) CLAMP AL
F1199  ; CONNECTOR CLAMP(4P-10S) UNCLAMP
F1200  ; CONNECTOR CLAMP(4P-10S) FWD ALAR
F1201  ; CONNECTOR CLAMP(4P-10S) BWD ALAR
F1202  ; CONNECTOR CLAMP(4P-10S-S) FWD AL
F1203  ; CONNECTOR CLAMP(4P-10S-S) BWD AL
F1204  ; CONNECTOR CLAMP(4P-10S-R) FWD AL
F1205  ; CONNECTOR CLAMP(4P-10S-R) BWD AL
F1206  ; BUS BAR CLEANING(FRONT) UP_4P AL
F1207  ; BUS BAR CLEANING(FRONT) DOWN_4P
F1208  ; BUS BAR CLEANING(REAR)  UP_4P AL
F1209  ; BUSBAR CLEANING(REAR) DOWN_4P AL
F1210  ; BUSBAR CHECK#1(FRONT)FWD_4P ALA
F1211  ; BUSBAR CHECK#1(FRONT)BWD_4P ALA
F1212  ; BUSBAR CHECK#2(FRONT)FWD_4P ALA
F1213  ; BUSBAR CHECK#2(FRONT)BWD_4P ALA
F1214  ; BUSBAR CHECK#3(FRONT)FWD_4P ALA
F1215  ; BUSBAR CHECK#3(FRONT)BWD_4P ALA
F1216  ; BUSBAR CHECK#4(FRONT)FWD_4P ALA
F1217  ; BUSBAR CHECK#4(FRONT)BWD_4P ALA
F1218  ; BUSBAR CHECK#5(FRONT)FWD_4P ALA
F1219  ; BUSBAR CHECK#5(FRONT)BWD_4P ALA
F1220  ; BUSBAR CHECK#6(FRONT)FWD_4P ALA
F1221  ; BUSBAR CHECK#6(FRONT)BWD_4P ALA
F1222  ; BUSBAR CHECK#7(FRONT)FWD_4P ALA
F1223  ; BUSBAR CHECK#7(FRONT)BWD_4P ALA
F1224  ; BUSBAR CHECK#8(FRONT)FWD_4P ALA
F1225  ; BUSBAR CHECK#8(FRONT)BWD_4P ALA
F1226  ; BUSBAR CHECK#9(FRONT)FWD_4P ALA
F1227  ; BUSBAR CHECK#9(FRONT)BWD_4P ALA
F1228  ; BUSBAR CHECK#10(FRONT)FWD_4P ALA
F1229  ; BUSBAR CHECK#10(FRONT)BWD_4P ALA
F1230  ; BUSBAR CHECK#1(REAR)FWD_4P ALA
F1231  ; BUSBAR CHECK#1(REAR)BWD_4P ALA
F1232  ; BUSBAR CHECK#2(REAR)FWD_4P ALA
F1233  ; BUSBAR CHECK#2(REAR)BWD_4P ALA
F1234  ; BUSBAR CHECK#3(REAR)FWD_4P ALA
F1235  ; BUSBAR CHECK#3(REAR)BWD_4P ALA
F1236  ; BUSBAR CHECK#4(REAR)FWD_4P ALA
F1237  ; BUSBAR CHECK#4(REAR)BWD_4P ALA
F1238  ; BUSBAR CHECK#5(REAR)FWD_4P ALA
F1239  ; BUSBAR CHECK#5(REAR)BWD_4P ALA
F1240  ; BUSBAR CHECK#6(REAR)FWD_4P ALA
F1241  ; BUSBAR CHECK#6(REAR)BWD_4P ALA
F1242  ; BUSBAR CHECK#7(REAR)FWD_4P ALA
F1243  ; BUSBAR CHECK#7(REAR)BWD_4P ALA
F1244  ; BUSBAR CHECK#8(REAR)FWD_4P ALA
F1245  ; BUSBAR CHECK#8(REAR)BWD_4P ALA
F1246  ; BUSBAR CHECK#9(REAR)FWD_4P ALA
F1247  ; BUSBAR CHECK#9(REAR)BWD_4P ALA
F1248  ; BUSBAR CHECK#10(REAR)FWD_4P ALA
F1249  ; BUSBAR CHECK#10(REAR)BWD_4P ALA
F1260  ; WORK UNLOAD4P10S/4P8S/2P18SFWD A
F1261  ; WORK UNLOAD4P10S/4P8S/2P18SBWD A
F1262  ; WORK UNLOAD4P10S/4P8S/2P18S CL A
F1263  ; WORK UNLOAD4P10S/4P8S/2P18SUCL A
F1264  ; WORK    UNLOAD  4P10S   CLAMP AL
F1265  ; WORK UNLOAD  4P10S UNCLAMP AL
F1266  ; WORK UNLOAD  4P8S  CLAMP AL
F1267  ; WORK UNLOAD  4P8S UNCLAMP AL
F1268  ; WORK UNLOAD  2P18S CLAMP AL
F1269  ; WORK UNLOAD  2P18S UNCLAMP AL
F1270  ; WORK UNLOAD  2P12S CLAMP AL
F1271  ; WORK  UNLOAD  2P12S UNCLAMP AL
F1272  ; WORK UNLOAD TURNING UNIT TURN AL
F1273  ; WORK UNLOAD TURNING RETURN AL
F1280  ; AOI 3D UPPER UNIT1 1-1,4 CL AL
F1281  ; AOI 3D UPPER UNIT1 1-1,4 UCL AL
F1282  ; AOI 3D UPPER UNIT1 1-2,3 CL AL
F1283  ; AOI 3D UPPER UNIT1 1-2,3 UCL AL
F1284  ; AOI 3D UPPER UNIT2 2-1 CL AL
F1285  ; AOI 3D UPPER UNIT2 2-1 UCL AL
F1286  ; AOI 3D UPPER UNIT2 2-2 CL AL
F1287  ; AOI 3D UPPER UNIT2 2-2 UCL AL
F1288  ; AOI 3D UPPER UNIT2 2-3 CL AL
F1289  ; AOI 3D UPPER UNIT2 2-3 UCL AL
F1290  ; AOI 3D UPPER UNIT2 2-4 CL AL
F1291  ; AOI 3D UPPER UNIT2 2-4 UCL AL
F1292  ; AOI 3D SIDE UNIT1 3-1,3 CL AL
F1293  ; AOI 3D SIDE UNIT1 3-1,3 UCL AL
F1294  ; AOI 3D SIDE UNIT1 3-2,4 CL AL
F1295  ; AOI 3D SIDE UNIT1 3-2,4 UCL AL
F1296  ; AOI 3D SIDE UNIT2 4-2,5 CL AL
F1297  ; AOI 3D SIDE UNIT2 4-2,5 UCL AL
F1298  ; AOI 3D SIDE UNIT2 4-1,4 CL AL
F1299  ; AOI 3D SIDE UNIT2 4-1,4 UCL AL
F1300  ; AOI 3D SIDE UNIT2 4-3,6 CL AL
F1301  ; AOI 3D SIDE UNIT2 4-3,6 UCL AL
F1302  ; AOI 3D SCANNER FRONT UP AL
F1303  ; AOI 3D SCANNER FRONT DN AL
F1304  ; AOI 3D SCANNER REAR UP AL
F1305  ; AOI 3D SCANNER REAR DN AL
D5600.0  ; 비젼2.출력완료
D6117.3  ; AX1.SV.HR.REQ
D6117.4  ; AX1.SV.HR.END
D6117.F  ; AX1.STATUS.POSITION.END
D6217.3  ; AX2.STATUS.HR.REQ
D6217.4  ; AX2.STATUS.HR.END
D6217.F  ; AX2.STATUS.POSITION.END
D7527.D  ; AX15.STATUS.ALARM
D7527.E  ; AX15.STATUS
D8091.0  ; HMI->PLC, HMI READY (1SEC)
